RoboDK station: Proyecto 1.rdk

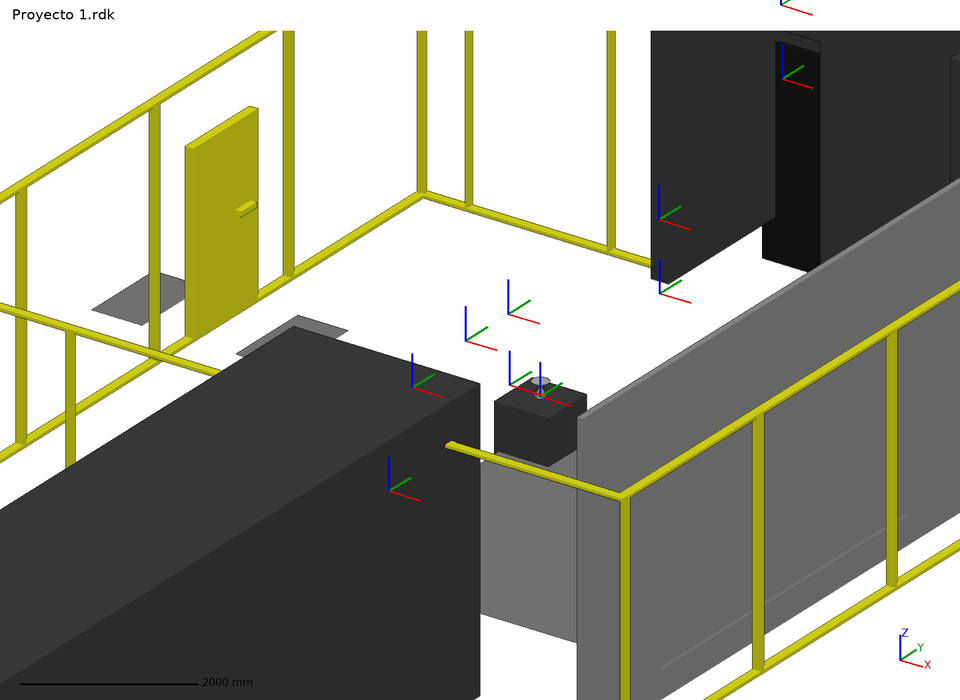
[picture v0: the station drawn from its stored meshes, robots at their saved joint values, targets as dots, program paths as lines]
Station Proyecto (saved by RoboDK 5.8.0). Poses are relative to the parent item; angles as X-Y-Z fixed-axis rotations.
Station parameters (name, value as stored): ColorElegido1, 1, ColorElegido2, 0, Robot1Operando, False, Robot2Operando, False
  - frame ABB IRB 580/12S_2 Base at (840.91, -2530.54, -390.83) mm
    - robot ABB IRB 580/12S 2 (model ABB IRB 580/12S): 6 axes, payload 12 kg, reach 2200 mm, repeatability 0.3 mm, weight 630 kg
        joint limits [-150, -70, -145, -360, -360, -720] to [150, 75, 145, 360, 360, 720]; home [0, 0, 0, 0, 0, 0]; saved at [0, 0, 0, 0, 0, 0]
      - tool TCP2, TCP at (0, -60, 0) mm, geometry from tinker.obj
        - object Herramienta at (0, 0, 0) mm, size 146.3 x 145.2 x 132 mm
        - object Cono at (0, 0, 0) mm, size 720 x 720 x 1182 mm
    - target Pintura21_1 (Cartesian target) at (1116.43, -38.64, 1773.81) mm, rotated rx 90 ry 0 rz 90 deg; joints [-2.419, -0.48, -16.124, 290.45, -28.618, -536.505] of ABB IRB 580/12S 2
    - target Pintura21_2 (Cartesian target) at (1117.91, -195.96, 1412.45) mm, rotated rx 90 ry 89.87 rz 90 deg; joints [-12.073, -6.734, 4.701, 191.643, 22.666, -570.657] of ABB IRB 580/12S 2
    - target Pintura21_3 (Cartesian target) at (1129.28, -196.63, 1042.61) mm, rotated rx 90 ry 89.87 rz 90 deg; joints [-11.969, -2.749, 25.87, 85.216, -50.511, -405.588] of ABB IRB 580/12S 2
    - target Pintura21_4 (Cartesian target) at (1138.7, -115.95, 957.64) mm, rotated rx 176.43 ry 87.92 rz 176.43 deg; joints [-7.055, -0.911, 30.503, 97.258, -52.14, -415.495] of ABB IRB 580/12S 2
    - target Pintura21_5 (Cartesian target) at (1212.31, 299.06, 873.56) mm, rotated rx 176.43 ry 87.92 rz 176.43 deg; joints [16.482, 10.653, 34.896, 146.51, -65.633, -445.211] of ABB IRB 580/12S 2
    - target Pintura21_6 (Cartesian target) at (1200.67, 359.89, 940.4) mm, rotated rx 176.43 ry 87.92 rz 176.43 deg; joints [19.809, 9.031, 31.023, 153.043, -62.201, -454.44] of ABB IRB 580/12S 2
    - target Pintura21_7 (Cartesian target) at (1202.62, 320.47, 971.04) mm, rotated rx 176.43 ry 87.92 rz 176.44 deg; joints [17.751, 7.276, 29.371, 149.237, -57.611, -455.624] of ABB IRB 580/12S 2
    - target Pintura21_8 (Cartesian target) at (1198.4, 183.42, 1272.89) mm, rotated rx 176.44 ry 87.92 rz 176.44 deg; joints [10.425, -0.652, 12.385, 146.399, -25.574, -483.886] of ABB IRB 580/12S 2
    - target Pintura21_9 (Cartesian target) at (1206.42, -176.13, 1230.65) mm, rotated rx 176.44 ry 87.92 rz 176.44 deg; joints [-9.943, 0.129, 14.76, -297.067, -28.151, -41.06] of ABB IRB 580/12S 2
    - target Pintura21_11 (Cartesian target) at (1119.11, -118.32, 1755.25) mm, rotated rx 90 ry 0 rz 90 deg; joints [-7.349, -0.419, -14.975, -51.416, -29.231, -193.501] of ABB IRB 580/12S 2
    - target Pintura21_13 (Cartesian target) at (939.03, -30.25, 1268.55) mm, rotated rx 90 ry 0 rz 90 deg; joints [-2.35, -24.007, 9.647, 83.365, -17.35, -339.315] of ABB IRB 580/12S 2
    - target Pintura21_14 (Cartesian target) at (920.1, -30.25, 1198.47) mm, rotated rx 136.9 ry 0 rz 90 deg; joints [-2.214, -19.899, 6.371, 304.189, -74.383, -511.521] of ABB IRB 580/12S 2
    - target Pintura21_15 (Cartesian target) at (812.29, -30.26, 846.49) mm, rotated rx 90 ry 0 rz 90 deg; joints [-2.837, -28.076, 32.69, 109.612, -58.975, -330.737] of ABB IRB 580/12S 2
    - target Pintura21_16 (Cartesian target) at (926.41, -30.26, 768.39) mm, rotated rx 73.79 ry 0 rz 90 deg; joints [-2.365, -7.019, 46.401, 147.807, -130.027, -297.801] of ABB IRB 580/12S 2
    - target Pintura21_17 (Cartesian target) at (1001.88, -30.25, 1480.86) mm, rotated rx 90 ry 0 rz 90 deg; joints [-2.165, -17.09, -0.641, 345.133, -3.937, -611.896] of ABB IRB 580/12S 2
    - target Pintura21_18 (Cartesian target) at (1001.88, -86.68, 1480.86) mm, rotated rx 90 ry 0 rz 90 deg; joints [-6.183, -16.757, -0.573, 359.165, -10.836, -620.25] of ABB IRB 580/12S 2
    - target Pintura21_19 (Cartesian target) at (1001.88, 52.48, 1480.86) mm, rotated rx 90 ry 0 rz 90 deg; joints [3.753, -16.997, -0.622, 192.113, -6.634, -456.698] of ABB IRB 580/12S 2
    - target Pintura21_20 (Cartesian target) at (1119.11, 44.39, 1755.25) mm, rotated rx 90 ry 0 rz 90 deg; joints [2.77, -0.951, -14.979, 270.402, -26.712, -518.755] of ABB IRB 580/12S 2
    - target Pintura21_21 (Cartesian target) at (1124.85, -28.64, 1773.81) mm, rotated rx 90 ry 0 rz 90 deg; joints [-1.777, 0.178, -16.122, 288.115, -28.472, -534.383] of ABB IRB 580/12S 2
    - target Pintura21_22 (Cartesian target) at (1118.79, 126.71, 1413.18) mm, rotated rx 90 ry 89.87 rz 90 deg; joints [7.867, -7.637, 4.583, 156.485, -15.894, -502.993] of ABB IRB 580/12S 2
    - target Pintura21_23 (Cartesian target) at (1111.66, 131.29, 1043.35) mm, rotated rx 90 ry 89.87 rz 90 deg; joints [8.211, -5.18, 25.707, 128.372, -47.85, -446.42] of ABB IRB 580/12S 2
    - target Pintura21_24 (Cartesian target) at (1116.6, 63.98, 964.01) mm, rotated rx 176.43 ry 87.92 rz 176.43 deg; joints [3.999, -3.356, 30.056, 119.508, -50.327, -436.143] of ABB IRB 580/12S 2
    - target Pintura21_25 (Cartesian target) at (1115.8, -383.46, 874.62) mm, rotated rx 176.43 ry 87.92 rz 176.43 deg; joints [-22.756, 5.765, 35.359, 83.262, -72.027, -389.304] of ABB IRB 580/12S 2
    - target Pintura21_26 (Cartesian target) at (1117.76, -430.8, 936.7) mm, rotated rx 176.43 ry 87.92 rz 176.44 deg; joints [-25.185, 5.256, 31.592, 75.5, -68.929, -384.335] of ABB IRB 580/12S 2
    - target Pintura21_27 (Cartesian target) at (1119.97, -379.27, 974.92) mm, rotated rx 176.43 ry 87.92 rz 176.44 deg; joints [-22.441, 2.586, 29.434, 74.391, -62.633, -387.628] of ABB IRB 580/12S 2
    - target Pintura21_28 (Cartesian target) at (1116.07, -255.92, 1270.03) mm, rotated rx 176.44 ry 87.92 rz 176.44 deg; joints [-15.636, -5.898, 12.34, 45.798, -32.699, -380.627] of ABB IRB 580/12S 2
    - target Pintura21_29 (Cartesian target) at (1113.24, 90.52, 1231.62) mm, rotated rx 176.44 ry 87.92 rz 176.44 deg; joints [5.669, -8.476, 14.275, -235.173, -23.506, -104.543] of ABB IRB 580/12S 2
    - target Pintura21_31 (Cartesian target) at (1117.02, 44.26, 1802.52) mm, rotated rx 90 ry 0 rz 90 deg; joints [2.768, 0.768, -17.925, -85.757, -31.888, -158.337] of ABB IRB 580/12S 2
    - target Pintura21_32 (Cartesian target) at (1119.85, 42.84, 1430.58) mm, rotated rx 90 ry 0 rz 90 deg; joints [2.672, -8.043, 3.565, 130.069, -7.77, -393.618] of ABB IRB 580/12S 2
    - target Pintura21_33 (Cartesian target) at (1113.28, 42.84, 1211.75) mm, rotated rx 90 ry 0 rz 90 deg; joints [2.691, -8.559, 15.797, 111.388, -28.118, -357.829] of ABB IRB 580/12S 2
    - target Pintura21_35 (Cartesian target) at (1350.01, 9.08, 882.74) mm, rotated rx 89.34 ry 0 rz 90 deg; joints [0.453, 17.806, 33.6, 116.92, -61.793, -334.561] of ABB IRB 580/12S 2
    - target Pintura21_34 (Cartesian target) at (1116.39, 45.51, 954.3) mm, rotated rx 78.25 ry 0 rz 90 deg; joints [2.836, -1.144, 33.638, 130.656, -84.724, -326.555] of ABB IRB 580/12S 2
    - target Pintura21_37 (Cartesian target) at (1116.39, -121.21, 954.3) mm, rotated rx 78.25 ry 0 rz 90 deg; joints [-7.514, -0.581, 33.644, 117.012, -85.786, -314.02] of ABB IRB 580/12S 2
    - target Pintura21_36 (Cartesian target) at (1350.01, -80.25, 882.74) mm, rotated rx 89.34 ry 0 rz 90 deg; joints [-3.998, 18.014, 33.552, 109.165, -62.094, -327.854] of ABB IRB 580/12S 2
    - target Pintura21_38 (Cartesian target) at (1113.28, -117.77, 1211.75) mm, rotated rx 90 ry 0 rz 90 deg; joints [-7.362, -8.006, 15.852, 77.337, -30.649, -323.061] of ABB IRB 580/12S 2
    - target Pintura21_39 (Cartesian target) at (1119.85, -118.25, 1430.58) mm, rotated rx 90 ry 0 rz 90 deg; joints [-7.339, -7.506, 3.615, 31.944, -14.28, -290.459] of ABB IRB 580/12S 2
    - target Pintura21_40 (Cartesian target) at (1117.02, -107.51, 1806.84) mm, rotated rx 90 ry 0 rz 90 deg; joints [-6.699, 1.387, -18.207, -55.298, -34.096, -185.427] of ABB IRB 580/12S 2
    - target Pintura22_ 1 (Cartesian target) at (1067.59, 53.4, 1620.15) mm, rotated rx 90 ry 0 rz 90 deg; joints [3.529, -9.086, -7.399, -109.72, -14.309, -148.767] of ABB IRB 580/12S 2
    - target Pintura22_ 2 (Cartesian target) at (1067.59, -94.87, 1462.33) mm, rotated rx 90 ry 0 rz 90 deg; joints [-6.253, -11.629, 1.35, -343.29, -11.164, 82.371] of ABB IRB 580/12S 2
    - target Pintura22_ 3 (Cartesian target) at (1067.59, -259.05, 1472.63) mm, rotated rx 90 ry 0 rz 90 deg; joints [-16.656, -8.853, 1.108, -344.207, -29.317, 98.232] of ABB IRB 580/12S 2
    - target Pintura22_ 4 (Cartesian target) at (1067.59, -164.34, 1317.72) mm, rotated rx 90 ry 0 rz 90 deg; joints [-10.747, -11.653, 9.477, -308.746, -25.051, 58.48] of ABB IRB 580/12S 2
    - target Pintura22_ 5 (Cartesian target) at (1067.59, -224.35, 1182.9) mm, rotated rx 90 ry 0 rz 90 deg; joints [-14.526, -9.793, 17.29, -294.626, -39.656, 55.316] of ABB IRB 580/12S 2
    - target Pintura22_ 6 (Cartesian target) at (1067.59, -116.53, 976.77) mm, rotated rx 90 ry 0 rz 90 deg; joints [-7.665, -7.234, 29.47, -262.498, -54.333, 36.08] of ABB IRB 580/12S 2
    - target Pintura22_ 7 (Cartesian target) at (1067.59, 409.36, 931.57) mm, rotated rx 90 ry 0 rz 90 deg; joints [25.304, 1.291, 32.515, -197.036, -73.881, -2.213] of ABB IRB 580/12S 2
    - target Pintura22_ 8 (Cartesian target) at (1067.59, 392.2, 1026.01) mm, rotated rx 90 ry 0 rz 90 deg; joints [24.369, -2.136, 26.86, -197.594, -64.501, -11.838] of ABB IRB 580/12S 2
    - target Pintura22_ 9 (Cartesian target) at (1067.59, 142.88, 1343.15) mm, rotated rx 90 ry 0 rz 90 deg; joints [9.37, -11.934, 8.012, -211.33, -21.539, -40.301] of ABB IRB 580/12S 2
    - target Pintura22_ 10 (Cartesian target) at (1067.59, -173.83, 1323.16) mm, rotated rx 90 ry 0 rz 90 deg; joints [-11.352, -11.499, 9.193, -310.971, -25.542, 61.091] of ABB IRB 580/12S 2
    - target Pintura22_ 11 (Cartesian target) at (1067.59, 304.45, 953.34) mm, rotated rx 90 ry 0 rz 90 deg; joints [19.372, -2.728, 31.16, -208.004, -65.531, -0.952] of ABB IRB 580/12S 2
    - target Pintura22_ 12 (Cartesian target) at (1137.59, 91.18, 1914.93) mm, rotated rx 110 ry 0 rz 90 deg; joints [5.378, 27.347, -40.85, 26.853, 124.647, -412.723] of ABB IRB 580/12S 2
    - target Pintura22_ 13 (Cartesian target) at (1137.59, 61.18, 1574.93) mm, rotated rx 90 ry 0 rz 90 deg; joints [3.74, -4.471, -4.383, 45.334, 10.05, -323.719] of ABB IRB 580/12S 2
    - target Pintura22_ 14 (Cartesian target) at (1007.59, 0, 1514.93) mm, rotated rx 110 ry 0 rz 90 deg; joints [0, -13.823, -5.955, -70.786, -46.099, -160.785] of ABB IRB 580/12S 2
    - target Pintura22_ 15 (Cartesian target) at (787.59, 0, 1244.93) mm, rotated rx 120 ry 0 rz 90 deg; joints [0, -34.851, 1.653, -68.861, -50.543, -158.857] of ABB IRB 580/12S 2
    - target Pintura22_ 16 (Cartesian target) at (837.59, 0, 784.93) mm, rotated rx 70 ry 0 rz 90 deg; joints [0, -15.633, 44.703, -154.776, 137.797, -244.777] of ABB IRB 580/12S 2
    - target Pintura22_ 17 (Cartesian target) at (1017.59, 50, 784.93) mm, rotated rx 70 ry 0 rz 90 deg; joints [3.455, 0.951, 46.49, -156.092, 146.166, -252.224] of ABB IRB 580/12S 2
    - target Pintura22_ 18 (Cartesian target) at (1017.59, -50, 784.93) mm, rotated rx 70 ry 0 rz 90 deg; joints [-3.456, 0.951, 46.49, -163.171, 146.167, -247.04] of ABB IRB 580/12S 2
    - target Pintura22_ 19 (Cartesian target) at (1057.59, 100, 1214.93) mm, rotated rx 110 ry 0 rz 90 deg; joints [6.572, -12.248, 11.285, -117.423, -18.827, -135.333] of ABB IRB 580/12S 2
    - target Pintura22_ 20 (Cartesian target) at (1057.59, 100, 1304.93) mm, rotated rx 80 ry 0 rz 90 deg; joints [6.641, -12.97, 11.964, -236.168, -40.558, -0.039] of ABB IRB 580/12S 2
    - target Pintura22_ 21 (Cartesian target) at (1137.59, -88.82, 1914.93) mm, rotated rx 110 ry 0 rz 90 deg; joints [-5.239, 27.293, -40.823, 38.325, 124.527, -421.835] of ABB IRB 580/12S 2
    - target Pintura22_ 22 (Cartesian target) at (1137.59, -68.82, 1574.93) mm, rotated rx 90 ry 0 rz 90 deg; joints [-4.206, -4.428, -4.38, 129.57, 10.592, -408.096] of ABB IRB 580/12S 2
    - target Pintura22_ 23 (Cartesian target) at (1057.59, -100, 1214.93) mm, rotated rx 110 ry 0 rz 90 deg; joints [-6.572, -12.248, 11.285, 117.416, 18.825, -404.663] of ABB IRB 580/12S 2
    - target Pintura22_ 24 (Cartesian target) at (1057.59, -100, 1304.93) mm, rotated rx 80 ry 0 rz 90 deg; joints [-6.641, -12.97, 11.964, 236.165, 40.559, -539.963] of ABB IRB 580/12S 2
    - target Pintura22_ 25 (Cartesian target) at (1067.59, -66.6, 1630.15) mm, rotated rx 90 ry 0 rz 90 deg; joints [-4.398, -8.769, -7.95, -54.41, -15.863, -202.263] of ABB IRB 580/12S 2
    - target Pintura22_ 26 (Cartesian target) at (1067.59, 65.12, 1462.33) mm, rotated rx 90 ry 0 rz 90 deg; joints [4.301, -11.851, 1.318, -193.793, -7.847, -69.726] of ABB IRB 580/12S 2
    - target Pintura22_ 27 (Cartesian target) at (1067.59, 230.95, 1472.63) mm, rotated rx 90 ry 0 rz 90 deg; joints [14.935, -9.472, 1.04, -173.077, -26.255, -75.157] of ABB IRB 580/12S 2
    - target Pintura22_ 28 (Cartesian target) at (1067.59, 145.66, 1297.72) mm, rotated rx 90 ry 0 rz 90 deg; joints [9.549, -11.917, 10.56, -217.204, -24.89, -31.418] of ABB IRB 580/12S 2
    - target Pintura22_ 29 (Cartesian target) at (1067.59, 175.65, 1182.9) mm, rotated rx 90 ry 0 rz 90 deg; joints [11.468, -10.727, 17.175, -220.502, -36.246, -17.745] of ABB IRB 580/12S 2
    - target Pintura22_ 30 (Cartesian target) at (1067.59, 73.47, 976.77) mm, rotated rx 90 ry 0 rz 90 deg; joints [4.85, -7.64, 29.432, -237.875, -53.256, 13.804] of ABB IRB 580/12S 2
    - target Pintura22_ 31 (Cartesian target) at (1067.59, -420.64, 931.57) mm, rotated rx 90 ry 0 rz 90 deg; joints [-25.911, 1.686, 32.507, -280.163, -74.568, 66.389] of ABB IRB 580/12S 2
    - target Pintura22_ 32 (Cartesian target) at (1067.59, -477.8, 1006.02) mm, rotated rx 90 ry 0 rz 90 deg; joints [-28.891, 1.54, 28.051, -288.806, -71.996, 72.955] of ABB IRB 580/12S 2
    - target Pintura22_ 33 (Cartesian target) at (1067.59, -187.12, 1323.15) mm, rotated rx 90 ry 0 rz 90 deg; joints [-12.194, -11.273, 9.224, -312.414, -26.747, 63.467] of ABB IRB 580/12S 2
    - target Pintura22_ 34 (Cartesian target) at (1067.59, 96.17, 1323.16) mm, rotated rx 90 ry 0 rz 90 deg; joints [6.338, -12.498, 9.051, -226.848, -19.298, -26.794] of ABB IRB 580/12S 2
    - target Pintura22_ 35 (Cartesian target) at (1067.59, -325.55, 953.34) mm, rotated rx 90 ry 0 rz 90 deg; joints [-20.605, -2.127, 31.178, -277.633, -66.76, 58.537] of ABB IRB 580/12S 2
    - target Pintura22_ 36 (Cartesian target) at (1236.43, -90.2, 1853.81) mm, rotated rx 109.13 ry 0 rz 90 deg; joints [-4.929, 20.785, -28.819, 315.941, -90.742, -506.111] of ABB IRB 580/12S 2
    - target Pintura22_ 37 (Cartesian target) at (1012.5, -90.2, 1474.16) mm, rotated rx 90.64 ry 0 rz 90 deg; joints [-6.348, -15.932, -0.16, 357.376, -11.167, -618.246] of ABB IRB 580/12S 2
    - target Pintura22_ 38 (Cartesian target) at (1094.1, -119.86, 1001.32) mm, rotated rx 90.64 ry 0 rz 90 deg; joints [-7.65, -5.739, 28.002, 232.585, 50.499, -546.78] of ABB IRB 580/12S 2
    - target Pintura22_ 39 (Cartesian target) at (1389.03, -96.9, 885.54) mm, rotated rx 83 ry 0 rz 90 deg; joints [-4.66, 21.788, 33.785, 230.644, 75.314, -566.392] of ABB IRB 580/12S 2
    - target Pintura22_ 40 (Cartesian target) at (1389.03, 71.9, 885.55) mm, rotated rx 83 ry 0 rz 90 deg; joints [3.461, 21.655, 33.821, 243.013, 75.168, -576.616] of ABB IRB 580/12S 2
    - target Pintura22_ 41 (Cartesian target) at (1094.1, 98.81, 1001.32) mm, rotated rx 90.64 ry 0 rz 90 deg; joints [6.318, -5.957, 27.986, 262.69, 49.904, -572.808] of ABB IRB 580/12S 2
    - target Pintura22_ 42 (Cartesian target) at (1012.5, 114.28, 1474.16) mm, rotated rx 90.64 ry 0 rz 90 deg; joints [8.023, -15.687, -0.113, 191.161, -14.073, -449.577] of ABB IRB 580/12S 2
    - target Pintura22_ 43 (Cartesian target) at (1236.43, 75.05, 1853.81) mm, rotated rx 109.13 ry 0 rz 90 deg; joints [4.104, 20.635, -28.772, 304.34, -90.475, -495.607] of ABB IRB 580/12S 2
    - target Pintura22_ 44 (Cartesian target) at (1208.68, -23.31, 1762.17) mm, rotated rx 90.64 ry 0 rz 90 deg; joints [-1.326, 6.871, -15.851, 286.646, -29.056, -532.5] of ABB IRB 580/12S 2
    - target Pintura22_ 45 (Cartesian target) at (1286.9, -13.32, 1041.23) mm, rotated rx 90.64 ry 0 rz 90 deg; joints [-0.703, 8.327, 25.435, 106.626, -43.976, -340.184] of ABB IRB 580/12S 2
    - target Pintura22_ 46 (Cartesian target) at (1224.34, -13.32, 1041.93) mm, rotated rx 90.64 ry 0.07 rz 83.59 deg; joints [0.515, 3.407, 25.753, 125.206, -46.158, -355.175] of ABB IRB 580/12S 2
    - target Pintura22_ 47 (Cartesian target) at (1230.82, -13.31, 1620.47) mm, rotated rx 90.64 ry 0.07 rz 83.59 deg; joints [0.511, 4.181, -7.144, 235.62, -18.187, -491.147] of ABB IRB 580/12S 2
    - target Pintura22_ 48 (Cartesian target) at (1230.82, -13.31, 1620.47) mm, rotated rx 90.63 ry -0.13 rz 101.88 deg; joints [-3.038, 4.556, -7.162, 345.144, -29.508, -589.807] of ABB IRB 580/12S 2
    - target Pintura22_ 49 (Cartesian target) at (1224, -13.32, 1012.28) mm, rotated rx 90.63 ry -0.13 rz 101.88 deg; joints [-3.058, 4.47, 27.441, 216.544, 54.407, -535.823] of ABB IRB 580/12S 2
    - object peana at (0, 0, -390) mm, rotated rx 90 ry 0 rz 0 deg, size 750 x 750 x 750 mm, 998277249 curves, geometry from peana.obj
  - frame ABB IRB 580/12S_1 Base at (840.91, 429.46, -390.83) mm
    - robot ABB IRB 580/12S 1 (model ABB IRB 580/12S): 6 axes, payload 12 kg, reach 2200 mm, repeatability 0.3 mm, weight 630 kg
        joint limits [-150, -70, -145, -360, -360, -720] to [150, 75, 145, 360, 360, 720]; home [0, 0, 0, 0, 0, 0]; saved at [-2.419, -0.48, -16.124, 290.45, -28.618, -176.505]
      - tool TCP1, TCP at (0, 0, 0) mm, geometry from tinker.obj
        - object Herramienta at (0, 0, 0) mm, size 146.3 x 145.2 x 132 mm
    - target Pintura11_1 (Cartesian target) at (1116.43, -38.64, 1773.81) mm, rotated rx 90 ry 0 rz 90 deg; joints [-2.419, -0.48, -16.124, 290.45, -28.618, -536.505] of ABB IRB 580/12S 1
    - target Pintura11_2 (Cartesian target) at (1117.91, -195.96, 1412.45) mm, rotated rx 90 ry 89.87 rz 90 deg; joints [-12.073, -6.734, 4.701, 191.643, 22.666, -570.657] of ABB IRB 580/12S 1
    - target Pintura11_3 (Cartesian target) at (1129.28, -196.63, 1042.61) mm, rotated rx 90 ry 89.87 rz 90 deg; joints [-11.969, -2.749, 25.87, 85.216, -50.511, -405.588] of ABB IRB 580/12S 1
    - target Pintura11_4 (Cartesian target) at (1138.7, -115.95, 957.64) mm, rotated rx 176.43 ry 87.92 rz 176.43 deg; joints [-7.055, -0.911, 30.503, 97.258, -52.14, -415.495] of ABB IRB 580/12S 1
    - target Pintura11_5 (Cartesian target) at (1212.31, 299.06, 873.56) mm, rotated rx 176.43 ry 87.92 rz 176.43 deg; joints [16.482, 10.653, 34.896, 146.51, -65.633, -445.211] of ABB IRB 580/12S 1
    - target Pintura11_6 (Cartesian target) at (1200.67, 359.89, 940.4) mm, rotated rx 176.43 ry 87.92 rz 176.43 deg; joints [19.809, 9.031, 31.023, 153.043, -62.201, -454.44] of ABB IRB 580/12S 1
    - target Pintura11_7 (Cartesian target) at (1202.62, 320.47, 971.04) mm, rotated rx 176.43 ry 87.92 rz 176.44 deg; joints [17.751, 7.276, 29.371, 149.237, -57.611, -455.624] of ABB IRB 580/12S 1
    - target Pintura11_8 (Cartesian target) at (1198.4, 183.42, 1272.89) mm, rotated rx 176.44 ry 87.92 rz 176.44 deg; joints [10.425, -0.652, 12.385, 146.399, -25.574, -483.886] of ABB IRB 580/12S 1
    - target Pintura11_9 (Cartesian target) at (1206.42, -176.13, 1230.65) mm, rotated rx 176.44 ry 87.92 rz 176.44 deg; joints [-9.943, 0.129, 14.76, -297.067, -28.151, -41.06] of ABB IRB 580/12S 1
    - target Pintura11_11 (Cartesian target) at (1119.11, -118.32, 1755.25) mm, rotated rx 90 ry 0 rz 90 deg; joints [-7.349, -0.419, -14.975, -51.416, -29.231, -193.501] of ABB IRB 580/12S 1
    - target Pintura11_13 (Cartesian target) at (939.03, -30.25, 1268.55) mm, rotated rx 90 ry 0 rz 90 deg; joints [-2.35, -24.007, 9.647, 83.365, -17.35, -339.315] of ABB IRB 580/12S 1
    - target Pintura11_14 (Cartesian target) at (920.1, -30.25, 1198.47) mm, rotated rx 136.9 ry 0 rz 90 deg; joints [-2.214, -19.899, 6.371, 304.189, -74.383, -511.521] of ABB IRB 580/12S 1
    - target Pintura11_15 (Cartesian target) at (812.29, -30.26, 846.49) mm, rotated rx 90 ry 0 rz 90 deg; joints [-2.837, -28.076, 32.69, 109.612, -58.975, -330.737] of ABB IRB 580/12S 1
    - target Pintura11_16 (Cartesian target) at (926.41, -30.26, 768.39) mm, rotated rx 73.79 ry 0 rz 90 deg; joints [-2.365, -7.019, 46.401, 147.807, -130.027, -297.801] of ABB IRB 580/12S 1
    - target Pintura11_17 (Cartesian target) at (1001.88, -30.25, 1480.86) mm, rotated rx 90 ry 0 rz 90 deg; joints [-2.165, -17.09, -0.641, 345.133, -3.937, -611.896] of ABB IRB 580/12S 1
    - target Pintura11_18 (Cartesian target) at (1001.88, -86.68, 1480.86) mm, rotated rx 90 ry 0 rz 90 deg; joints [-6.183, -16.757, -0.573, 359.165, -10.836, -620.25] of ABB IRB 580/12S 1
    - target Pintura11_19 (Cartesian target) at (1001.88, 52.48, 1480.86) mm, rotated rx 90 ry 0 rz 90 deg; joints [3.753, -16.997, -0.622, 192.113, -6.634, -456.698] of ABB IRB 580/12S 1
    - target Pintura11_20 (Cartesian target) at (1119.11, 44.39, 1755.25) mm, rotated rx 90 ry 0 rz 90 deg; joints [2.77, -0.951, -14.979, 270.402, -26.712, -518.755] of ABB IRB 580/12S 1
    - target Pintura12_1 (Cartesian target) at (1067.59, 13.4, 1620.15) mm, rotated rx 90 ry 0 rz 90 deg; joints [0.887, -9.208, -7.413, -91.494, -13.034, -167.871] of ABB IRB 580/12S 1
    - target Pintura12_2 (Cartesian target) at (1067.59, -94.87, 1462.33) mm, rotated rx 90 ry 0 rz 90 deg; joints [-6.253, -11.629, 1.35, -343.29, -11.164, 82.371] of ABB IRB 580/12S 1
    - target Pintura12_3 (Cartesian target) at (1067.59, -259.05, 1472.63) mm, rotated rx 90 ry 0 rz 90 deg; joints [-16.656, -8.853, 1.108, -344.207, -29.317, 98.232] of ABB IRB 580/12S 1
    - target Pintura12_4 (Cartesian target) at (1067.59, -224.34, 1297.72) mm, rotated rx 90 ry 0 rz 90 deg; joints [-14.526, -10.541, 10.744, -311.194, -31.651, 65.963] of ABB IRB 580/12S 1
    - target Pintura12_5 (Cartesian target) at (1067.59, -224.35, 1182.9) mm, rotated rx 90 ry 0 rz 90 deg; joints [-14.526, -9.793, 17.29, -294.626, -39.656, 55.316] of ABB IRB 580/12S 1
    - target Pintura12_6 (Cartesian target) at (1067.59, -116.53, 976.77) mm, rotated rx 90 ry 0 rz 90 deg; joints [-7.665, -7.234, 29.47, -262.498, -54.333, 36.08] of ABB IRB 580/12S 1
    - target Pintura12_7 (Cartesian target) at (1067.59, 389.36, 931.57) mm, rotated rx 90 ry 0 rz 90 deg; joints [24.212, 0.61, 32.523, -199.021, -72.671, -1.681] of ABB IRB 580/12S 1
    - target Pintura12_8 (Cartesian target) at (1067.59, 382.2, 1006.01) mm, rotated rx 90 ry 0 rz 90 deg; joints [23.817, -1.941, 28.042, -199.018, -65.5, -9.384] of ABB IRB 580/12S 1
    - target Pintura12_9 (Cartesian target) at (1067.59, 122.88, 1323.15) mm, rotated rx 90 ry 0 rz 90 deg; joints [8.078, -12.217, 9.092, -219.336, -21.246, -32.553] of ABB IRB 580/12S 1
    - target Pintura12_10 (Cartesian target) at (1067.59, -173.83, 1323.16) mm, rotated rx 90 ry 0 rz 90 deg; joints [-11.352, -11.499, 9.193, -310.971, -25.542, 61.091] of ABB IRB 580/12S 1
    - target Pintura12_11 (Cartesian target) at (1067.59, 274.45, 953.34) mm, rotated rx 90 ry 0 rz 90 deg; joints [17.587, -3.524, 31.128, -211.447, -63.849, 0.455] of ABB IRB 580/12S 1
    - target Pintura12_37 (Cartesian target) at (1236.43, -90.2, 1853.81) mm, rotated rx 109.13 ry 0 rz 90 deg; joints [-4.929, 20.785, -28.819, 315.941, -90.742, -506.111] of ABB IRB 580/12S 1
    - target Pintura12_38 (Cartesian target) at (1012.5, -90.2, 1474.16) mm, rotated rx 90.64 ry 0 rz 90 deg; joints [-6.348, -15.932, -0.16, 357.376, -11.167, -618.246] of ABB IRB 580/12S 1
    - target Pintura12_39 (Cartesian target) at (1094.1, -119.86, 1001.32) mm, rotated rx 90.64 ry 0 rz 90 deg; joints [-7.65, -5.739, 28.002, 232.585, 50.499, -546.78] of ABB IRB 580/12S 1
    - target Pintura12_40 (Cartesian target) at (1389.03, -96.9, 885.54) mm, rotated rx 83 ry 0 rz 90 deg; joints [-4.66, 21.788, 33.785, 230.644, 75.314, -566.392] of ABB IRB 580/12S 1
    - target Pintura12_41 (Cartesian target) at (1389.03, 71.9, 885.55) mm, rotated rx 83 ry 0 rz 90 deg; joints [3.461, 21.655, 33.821, 243.013, 75.168, -576.616] of ABB IRB 580/12S 1
    - target Pintura12_42 (Cartesian target) at (1094.1, 98.81, 1001.32) mm, rotated rx 90.64 ry 0 rz 90 deg; joints [6.318, -5.957, 27.986, 262.69, 49.904, -572.808] of ABB IRB 580/12S 1
    - target Pintura12_43 (Cartesian target) at (1012.5, 114.28, 1474.16) mm, rotated rx 90.64 ry 0 rz 90 deg; joints [8.023, -15.687, -0.113, 191.161, -14.073, -449.577] of ABB IRB 580/12S 1
    - target Pintura12_44 (Cartesian target) at (1236.43, 75.05, 1853.81) mm, rotated rx 109.13 ry 0 rz 90 deg; joints [4.104, 20.635, -28.772, 304.34, -90.475, -495.607] of ABB IRB 580/12S 1
    - target Pintura12_45 (Cartesian target) at (1208.68, -23.31, 1762.17) mm, rotated rx 90.64 ry 0 rz 90 deg; joints [-1.326, 6.871, -15.851, 286.646, -29.056, -532.5] of ABB IRB 580/12S 1
    - target Pintura12_46 (Cartesian target) at (1286.9, -13.32, 1041.23) mm, rotated rx 90.64 ry 0 rz 90 deg; joints [-0.703, 8.327, 25.435, 106.626, -43.976, -340.184] of ABB IRB 580/12S 1
    - target Pintura12_47 (Cartesian target) at (1224.34, -13.32, 1041.93) mm, rotated rx 90.64 ry 0.07 rz 83.59 deg; joints [0.515, 3.407, 25.753, 125.206, -46.158, -355.175] of ABB IRB 580/12S 1
    - target Pintura12_48 (Cartesian target) at (1230.82, -13.31, 1620.47) mm, rotated rx 90.64 ry 0.07 rz 83.59 deg; joints [0.511, 4.181, -7.144, 235.62, -18.187, -491.147] of ABB IRB 580/12S 1
    - target Pintura12_49 (Cartesian target) at (1230.82, -13.31, 1620.47) mm, rotated rx 90.63 ry -0.13 rz 101.88 deg; joints [-3.038, 4.556, -7.162, 345.144, -29.508, -589.807] of ABB IRB 580/12S 1
    - target Pintura12_50 (Cartesian target) at (1224, -13.32, 1012.28) mm, rotated rx 90.63 ry -0.13 rz 101.88 deg; joints [-3.058, 4.47, 27.441, 216.544, 54.407, -535.823] of ABB IRB 580/12S 1
    - target Pintura11_21 (Cartesian target) at (1124.85, -18.64, 1773.81) mm, rotated rx 90 ry 0 rz 90 deg; joints [-1.157, 0.157, -16.122, 285.858, -28.374, -532.295] of ABB IRB 580/12S 1
    - target Pintura11_22 (Cartesian target) at (1118.79, 126.71, 1413.18) mm, rotated rx 90 ry 89.87 rz 90 deg; joints [7.867, -7.637, 4.583, 156.485, -15.894, -502.993] of ABB IRB 580/12S 1
    - target Pintura11_23 (Cartesian target) at (1111.66, 131.29, 1043.35) mm, rotated rx 90 ry 89.87 rz 90 deg; joints [8.211, -5.18, 25.707, 128.372, -47.85, -446.42] of ABB IRB 580/12S 1
    - target Pintura11_24 (Cartesian target) at (1116.6, 63.98, 964.01) mm, rotated rx 176.43 ry 87.92 rz 176.43 deg; joints [3.999, -3.356, 30.056, 119.508, -50.327, -436.143] of ABB IRB 580/12S 1
    - target Pintura11_25 (Cartesian target) at (1115.8, -383.46, 874.62) mm, rotated rx 176.43 ry 87.92 rz 176.43 deg; joints [-22.756, 5.765, 35.359, 83.262, -72.027, -389.304] of ABB IRB 580/12S 1
    - target Pintura11_26 (Cartesian target) at (1117.76, -430.8, 936.7) mm, rotated rx 176.43 ry 87.92 rz 176.44 deg; joints [-25.185, 5.256, 31.592, 75.5, -68.929, -384.335] of ABB IRB 580/12S 1
    - target Pintura11_27 (Cartesian target) at (1119.97, -379.27, 974.92) mm, rotated rx 176.43 ry 87.92 rz 176.44 deg; joints [-22.441, 2.586, 29.434, 74.391, -62.633, -387.628] of ABB IRB 580/12S 1
    - target Pintura11_28 (Cartesian target) at (1116.07, -255.92, 1270.03) mm, rotated rx 176.44 ry 87.92 rz 176.44 deg; joints [-15.636, -5.898, 12.34, 45.798, -32.699, -380.627] of ABB IRB 580/12S 1
    - target Pintura11_29 (Cartesian target) at (1113.24, 90.52, 1231.62) mm, rotated rx 176.44 ry 87.92 rz 176.44 deg; joints [5.669, -8.476, 14.275, -235.173, -23.506, -104.543] of ABB IRB 580/12S 1
    - target Pintura11_31 (Cartesian target) at (1117.02, 44.26, 1802.52) mm, rotated rx 90 ry 0 rz 90 deg; joints [2.768, 0.768, -17.925, -85.757, -31.888, -158.337] of ABB IRB 580/12S 1
    - target Pintura11_32 (Cartesian target) at (1119.85, 42.84, 1430.58) mm, rotated rx 90 ry 0 rz 90 deg; joints [2.672, -8.043, 3.565, 130.069, -7.77, -393.618] of ABB IRB 580/12S 1
    - target Pintura11_33 (Cartesian target) at (1113.28, 42.84, 1211.75) mm, rotated rx 90 ry 0 rz 90 deg; joints [2.691, -8.559, 15.797, 111.388, -28.118, -357.829] of ABB IRB 580/12S 1
    - target Pintura11_35 (Cartesian target) at (1350.01, 9.08, 882.74) mm, rotated rx 89.34 ry 0 rz 90 deg; joints [0.453, 17.806, 33.6, 116.92, -61.793, -334.561] of ABB IRB 580/12S 1
    - target Pintura11_34 (Cartesian target) at (1116.39, 45.51, 954.3) mm, rotated rx 78.25 ry 0 rz 90 deg; joints [2.836, -1.144, 33.638, 130.656, -84.724, -326.555] of ABB IRB 580/12S 1
    - target Pintura11_37 (Cartesian target) at (1116.39, -121.21, 954.3) mm, rotated rx 78.25 ry 0 rz 90 deg; joints [-7.514, -0.581, 33.644, 117.012, -85.786, -314.02] of ABB IRB 580/12S 1
    - target Pintura11_36 (Cartesian target) at (1350.01, -80.25, 882.74) mm, rotated rx 89.34 ry 0 rz 90 deg; joints [-3.998, 18.014, 33.552, 109.165, -62.094, -327.854] of ABB IRB 580/12S 1
    - target Pintura11_38 (Cartesian target) at (1113.28, -117.77, 1211.75) mm, rotated rx 90 ry 0 rz 90 deg; joints [-7.362, -8.006, 15.852, 77.337, -30.649, -323.061] of ABB IRB 580/12S 1
    - target Pintura11_39 (Cartesian target) at (1119.85, -118.25, 1430.58) mm, rotated rx 90 ry 0 rz 90 deg; joints [-7.339, -7.506, 3.615, 31.944, -14.28, -290.459] of ABB IRB 580/12S 1
    - target Pintura11_40 (Cartesian target) at (1117.02, -107.51, 1806.84) mm, rotated rx 90 ry 0 rz 90 deg; joints [-6.699, 1.387, -18.207, -55.298, -34.096, -185.427] of ABB IRB 580/12S 1
    - target Pintura12_13 (Cartesian target) at (1137.59, 91.18, 1934.93) mm, rotated rx 110 ry 0 rz 90 deg; joints [5.494, 17.782, -34.165, 36.405, 105.718, -401.654] of ABB IRB 580/12S 1
    - target Pintura12_14 (Cartesian target) at (1137.59, 61.18, 1574.93) mm, rotated rx 90 ry 0 rz 90 deg; joints [3.74, -4.471, -4.383, 45.334, 10.05, -323.719] of ABB IRB 580/12S 1
    - target Pintura12_15 (Cartesian target) at (1007.59, 0, 1514.93) mm, rotated rx 110 ry 0 rz 90 deg; joints [0, -13.823, -5.955, -70.786, -46.099, -160.785] of ABB IRB 580/12S 1
    - target Pintura12_16 (Cartesian target) at (787.59, 0, 1244.93) mm, rotated rx 120 ry 0 rz 90 deg; joints [0, -34.851, 1.653, -68.861, -50.543, -158.857] of ABB IRB 580/12S 1
    - target Pintura12_17 (Cartesian target) at (837.59, 0, 784.93) mm, rotated rx 70 ry 0 rz 90 deg; joints [0, -15.633, 44.703, -154.776, 137.797, -244.777] of ABB IRB 580/12S 1
    - target Pintura12_18 (Cartesian target) at (1017.59, 50, 784.93) mm, rotated rx 70 ry 0 rz 90 deg; joints [3.455, 0.951, 46.49, -156.092, 146.166, -252.224] of ABB IRB 580/12S 1
    - target Pintura12_19 (Cartesian target) at (1017.59, -50, 784.93) mm, rotated rx 70 ry 0 rz 90 deg; joints [-3.456, 0.951, 46.49, -163.171, 146.167, -247.04] of ABB IRB 580/12S 1
    - target Pintura12_20 (Cartesian target) at (1057.59, 100, 1214.93) mm, rotated rx 110 ry 0 rz 90 deg; joints [6.572, -12.248, 11.285, -117.423, -18.827, -135.333] of ABB IRB 580/12S 1
    - target Pintura12_21 (Cartesian target) at (1057.59, 100, 1304.93) mm, rotated rx 80 ry 0 rz 90 deg; joints [6.641, -12.97, 11.964, -236.168, -40.558, -0.039] of ABB IRB 580/12S 1
    - target Pintura12_22 (Cartesian target) at (1137.59, -88.82, 1934.93) mm, rotated rx 110 ry 0 rz 90 deg; joints [-5.352, 17.754, -34.157, 48.973, 105.665, -412.663] of ABB IRB 580/12S 1
    - target Pintura12_23 (Cartesian target) at (1137.59, -68.82, 1574.93) mm, rotated rx 90 ry 0 rz 90 deg; joints [-4.206, -4.428, -4.38, 129.57, 10.592, -408.096] of ABB IRB 580/12S 1
    - target Pintura12_24 (Cartesian target) at (1057.59, -100, 1214.93) mm, rotated rx 110 ry 0 rz 90 deg; joints [-6.572, -12.248, 11.285, 117.416, 18.825, -404.663] of ABB IRB 580/12S 1
    - target Pintura12_25 (Cartesian target) at (1057.59, -100, 1304.93) mm, rotated rx 80 ry 0 rz 90 deg; joints [-6.641, -12.97, 11.964, 236.165, 40.559, -539.963] of ABB IRB 580/12S 1
    - target Pintura12_26 (Cartesian target) at (1067.59, -26.6, 1760.15) mm, rotated rx 90 ry 0 rz 90 deg; joints [-1.76, -4.948, -15.437, -72.183, -27.257, -175.112] of ABB IRB 580/12S 1
    - target Pintura12_27 (Cartesian target) at (1067.59, 65.12, 1462.33) mm, rotated rx 90 ry 0 rz 90 deg; joints [4.301, -11.851, 1.318, -193.793, -7.847, -69.726] of ABB IRB 580/12S 1
    - target Pintura12_28 (Cartesian target) at (1067.59, 230.95, 1472.63) mm, rotated rx 90 ry 0 rz 90 deg; joints [14.935, -9.472, 1.04, -173.077, -26.255, -75.157] of ABB IRB 580/12S 1
    - target Pintura12_29 (Cartesian target) at (1067.59, 145.66, 1297.72) mm, rotated rx 90 ry 0 rz 90 deg; joints [9.549, -11.917, 10.56, -217.204, -24.89, -31.418] of ABB IRB 580/12S 1
    - target Pintura12_30 (Cartesian target) at (1067.59, 175.65, 1182.9) mm, rotated rx 90 ry 0 rz 90 deg; joints [11.468, -10.727, 17.175, -220.502, -36.246, -17.745] of ABB IRB 580/12S 1
    - target Pintura12_31 (Cartesian target) at (1067.59, 73.47, 976.77) mm, rotated rx 90 ry 0 rz 90 deg; joints [4.85, -7.64, 29.432, -237.875, -53.256, 13.804] of ABB IRB 580/12S 1
    - target Pintura12_32 (Cartesian target) at (1067.59, -420.64, 931.57) mm, rotated rx 90 ry 0 rz 90 deg; joints [-25.911, 1.686, 32.507, -280.163, -74.568, 66.389] of ABB IRB 580/12S 1
    - target Pintura12_33 (Cartesian target) at (1067.59, -477.8, 1006.02) mm, rotated rx 90 ry 0 rz 90 deg; joints [-28.891, 1.54, 28.051, -288.806, -71.996, 72.955] of ABB IRB 580/12S 1
    - target Pintura12_34 (Cartesian target) at (1067.59, -187.12, 1323.15) mm, rotated rx 90 ry 0 rz 90 deg; joints [-12.194, -11.273, 9.224, -312.414, -26.747, 63.467] of ABB IRB 580/12S 1
    - target Pintura12_35 (Cartesian target) at (1067.59, 96.17, 1323.16) mm, rotated rx 90 ry 0 rz 90 deg; joints [6.338, -12.498, 9.051, -226.848, -19.298, -26.794] of ABB IRB 580/12S 1
    - target Pintura12_36 (Cartesian target) at (1067.59, -325.55, 953.34) mm, rotated rx 90 ry 0 rz 90 deg; joints [-20.605, -2.127, 31.178, -277.633, -66.76, 58.537] of ABB IRB 580/12S 1
    - object peana at (0, 0, -390) mm, rotated rx 90 ry 0 rz 0 deg, size 750 x 750 x 750 mm, 998277249 curves, geometry from peana.obj
  - frame Frame Grua at (2500, -3400.54, 2300) mm
    - object grua at (0, 0, 0) mm, rotated rx 90 ry 0 rz 0 deg, size 0 x 0 x 0 mm, 1044167869 curves, geometry from grua.obj
  - frame Frame 8 at (0, -870.54, 0) mm
    - object Fabrica 1 at (0, 0, -1030) mm, rotated rx 90 ry 0 rz 0 deg
    - object Pasillo 2 at (4600, 16100, -1460) mm, rotated rx 90 ry 0 rz 90 deg, size 20643.2 x 3904.4 x 2560.3 mm, geometry from Pasillo 2.obj
    - object Pasillo 2 at (500, 16100, -1460) mm, rotated rx 90 ry 0 rz 90 deg, size 20643.2 x 3904.4 x 2560.3 mm, geometry from Pasillo 2.obj
    - object Pasillo 2 at (2500, -14400, -1460) mm, rotated rx 90 ry 0 rz 90 deg, size 20643.2 x 3904.4 x 2560.3 mm, geometry from Pasillo 2.obj
    - object Valla 2 at (-200, 0, 0) mm, rotated rx 0 ry 0 rz -90 deg, size 120 x 3276.4 x 2628 mm, geometry from Valla 2.obj
    - object Valla 2 at (1450, -8420, 0) mm, size 120 x 3276.4 x 2628 mm, geometry from Valla 2.obj
    - object Valla 2 at (1450, -5800, 0) mm, size 120 x 3276.4 x 2628 mm, geometry from Valla 2.obj
    - object Valla 2 at (2180, -1330, 0) mm, rotated rx 0 ry 0 rz 10 deg, size 120 x 3276.4 x 2628 mm, geometry from Valla 2.obj
    - object Valla 2 at (1450, -3180, 0) mm, size 120 x 3276.4 x 2628 mm, geometry from Valla 2.obj
    - object Valla 2 at (-5180, 0, 0) mm, rotated rx 0 ry 0 rz -90 deg, size 120 x 3276.4 x 2628 mm, geometry from Valla 2.obj
    - object Valla 2 at (-8660, -8420, 0) mm, size 120 x 3276.4 x 2628 mm, geometry from Valla 2.obj
    - object Valla 2 at (-7800, 0, 0) mm, rotated rx 0 ry 0 rz -90 deg, size 120 x 3276.4 x 2628 mm, geometry from Valla 2.obj
    - object Valla 2 at (-8660, -5800, 0) mm, size 120 x 3276.4 x 2628 mm, geometry from Valla 2.obj
    - object Valla 3 at (-3960, 1910, -1030) mm, rotated rx 90 ry 0 rz 0 deg, size 284.8 x 3276.4 x 2628 mm, geometry from Valla 3.obj
    - object Valla 2 at (-7760, 10540, 0) mm, rotated rx 0 ry 0 rz -90 deg, size 120 x 3276.4 x 2628 mm, geometry from Valla 2.obj
    - object Valla 2 at (-8660, -560, 0) mm, size 120 x 3276.4 x 2628 mm, geometry from Valla 2.obj
    - object Valla 2 at (-7110, 10540, 0) mm, rotated rx 0 ry 0 rz -90 deg, size 120 x 3276.4 x 2628 mm, geometry from Valla 2.obj
    - object IRONLINELOGOChasis at (-460, 0, 0) mm, size 4826 x 4699 x 0 mm, 1046087008 curves, geometry from IRONLINELOGOChasis.png
    - object pared at (-500, 0, 0) mm, size 83.4 x 3742.7 x 4117 mm, geometry from pared.obj
    - object pared at (-500, 0, 0) mm, size 83.4 x 3742.7 x 4117 mm, geometry from pared.obj
    - object IronLineFUll text at (0, 0, 0) mm, size 5022.9 x 2070.1 x 0 mm, 1046086528 curves, geometry from IronLineFUll text.png
    - object pared at (0, 0, 0) mm, size 2495.2 x 55.6 x 2744.6 mm
    - object pared at (1960, -13550, 0) mm, size 2495.2 x 55.6 x 2744.6 mm
    - object pared at (4100, 0, 0) mm, size 2495.2 x 55.6 x 2744.6 mm
    - object Flecha at (-330, 0, 0) mm, size 1219.2 x 693.6 x 0 mm, 1046083728 curves, geometry from Flecha.png
    - object Flecha at (-7590, 3760, 0) mm, rotated rx 0 ry 0 rz -180 deg, size 1219.2 x 693.6 x 0 mm, 1046083728 curves, geometry from Flecha.png
    - object Ralla at (-1300, -160, -1020) mm
    - object pared at (13600, 0, 0) mm, size 83.4 x 3742.7 x 4117 mm, geometry from pared.obj
  - frame Frame 6 at (2490.38, -2530.4, 1393.84) mm
    - object Chopper Frame AP203 2 at (-5, -165, -630) mm, rotated rx 0 ry -90 rz 0 deg
  - frame Frame C1 at (4518.72, 5642.83, 2280.87) mm
    - object Cilindro2 at (-60, 0, -830) mm, rotated rx 0 ry 4.5 rz 0 deg
  - frame Frame H1 at (2478.72, 415.5, 2280.87) mm
    - object Cilindro2 at (-60, 0, -830) mm, rotated rx 0 ry 4.5 rz 0 deg
  - frame Frame 4 at (4530.38, 5646.93, 1393.84) mm
    - object Chopper Frame AP203 1 at (-5, -165, -630) mm, rotated rx 0 ry -90 rz 0 deg
  - frame Frame 5 at (2485.91, 420, 1357.58) mm
    - object Frame cb 750 1 at (0, -127.82, -424.28) mm, rotated rx 90 ry -70 rz -90 deg
  - frame Frame C2 at (2478.72, -2534.5, 2280.87) mm
    - object Cilindro3 at (-60, 0, -830) mm, rotated rx 0 ry 4.5 rz 0 deg
  - frame Frame H2 at (448.72, 5708.5, 2280.87) mm
    - object Cilindro2 at (-60, 0, -830) mm, rotated rx 0 ry 4.5 rz 0 deg
  - frame Frame 7 at (455.92, 5713, 1357.58) mm
    - object Frame cb 750 2 at (0, -127.82, -424.28) mm, rotated rx 90 ry -70 rz -90 deg
  - folder Programas
    - Python program Honda11 (listed below)
    - Python program Honda12 (listed below)
    - Python program Chopper11 (listed below)
    - Python program Chopper12 (listed below)
    - Python program Honda21 (listed below)
    - Python program Honda22 (listed below)
    - Python program Chopper21 (listed below)
    - Python program Chopper22 (listed below)
    - Python program SprayOn (listed below)
    - Python program MoverHonda11 (listed below)
    - Python program MoverHonda12 (listed below)
    - Python program MoverChopper11 (listed below)
    - Python program MoverChopper12 (listed below)
    - Python program MoverHonda21 (listed below)
    - Python program MoverHonda22 (listed below)
    - Python program MoverChopper21 (listed below)
    - Python program MoverChopper22 (listed below)
    - Python program MoverChopper11Final (listed below)
    - Python program MoverChopper12Final (listed below)
    - Python program MoverHonda11Final (listed below)
    - Python program MoverHonda12Final (listed below)
    - Python program MoverChopper21Final (listed below)
    - Python program MoverChopper22Final (listed below)
    - Python program MoverHonda21Final (listed below)
    - Python program MoverHonda22Final (listed below)
  - program Honda1Robot1 (3 instructions, listed below)
  - program Honda2Robot1 (3 instructions, listed below)
  - program Honda1Robot2 (3 instructions, listed below)
  - program Honda2Robot2 (3 instructions, listed below)
  - program Chopper1Robot1 (3 instructions, listed below)
  - program Chopper2Robot1 (3 instructions, listed below)
  - program Chopper1Robot2 (3 instructions, listed below)
  - program Chopper2Robot2 (3 instructions, listed below)

--- Python program Honda11 ---
from robodk.robolink import *  # API de RoboDK
from robodk.robomath import *  # Funciones matemáticas
import time
import math

# Inicializar conexión con RoboDK
RDK = Robolink()

# Borrar las partículas de pintura previas
RDK.Spray_Clear()

# Comprobar si estamos en modo simulación
if RDK.RunMode() != RUNMODE_SIMULATE:
    raise Exception('El robot no está en modo simulación')

# Obtener el robot
robot = RDK.Item('ABB IRB 580/12S 1', ITEM_TYPE_ROBOT)
if not robot.Valid():
    raise Exception('Robot "ABB IRB 580/12S 1" no encontrado')

# Establecer herramienta activa (TCP1)
tool = RDK.Item('TCP1', ITEM_TYPE_TOOL)
if not tool.Valid():
    raise Exception('Herramienta TCP1 no encontrada')
robot.setTool(tool)

# Obtener el objeto a pintar
honda = RDK.Item('Frame cb 750 1', ITEM_TYPE_OBJECT)
if not honda.Valid():
    raise Exception('Objeto "Frame cb 750 1" no encontrado')

# Obtener el sistema del gancho
frame6 = RDK.Item('Frame H1', ITEM_TYPE_FRAME)
if not frame6.Valid():
    raise Exception('Sistema "Frame H1" no encontrado')

# Obtener el sistema de la honda
frame5 = RDK.Item('Frame 5', ITEM_TYPE_FRAME)
if not frame5.Valid():
    raise Exception('Sistema "Frame 5" no encontrado')



# -------------------------
# MAPEO DE COLORES
# -------------------------
colores_numericos = {
    0: [1.0, 0.0, 0.0],  # rojo
    1: [0.0, 0.0, 0.0],  # negro
    2: [0.0, 1.0, 0.0],  # verde
    3: [0.5, 0.5, 0.5],  # gris
    4: [1.0, 1.0, 1.0],  # blanco
    5: [1.0, 0.5, 0.0]   # naranja
}

# Obtener número desde variable global de RoboDK
valor_color = RDK.getParam('ColorElegido1')
if valor_color is None:
    valor_color = 0  # valor por defecto
valor_color = int(valor_color)

if valor_color not in colores_numericos:
    raise Exception(f'ColorElegido inválido: {valor_color}')
color_final = colores_numericos[valor_color]

# Color neutro inicial
color_inicial = [0.9, 0.9, 0.9]

# Activar pintado automático
options_command = "ELLYPSE PROJECT PARTICLE=SPHERE(4,10,1,1,0.5) STEP=3x3 RAND=2"
close_param = [0, 0, 0, 5, 0, 0, 0, 5, 0, color_final[0], color_final[1], color_final[2], 1]
far_param   = [0, 0, 2000, 500, 0, 2000, 0, 500, 2000, color_final[0], color_final[1], color_final[2], 0.2]
volume = Mat([close_param, far_param]).tr()
RDK.Spray_Add(tool, honda, options_command, volume)
RDK.Spray_SetState(SPRAY_ON)

# Establecer velocidades lentas
robot.setSpeed(50, 50)
robot.setAcceleration(50)

# Lista de nombres de targets
targets = [
    'Pintura11_1',
    'Pintura12_1',
    'Pintura12_4',
    'Pintura12_3',
    'Pintura12_2',
    'Pintura12_5',
    'Pintura12_6',
    'Pintura12_7',
    'Pintura12_8',
    'Pintura12_9',
    'Pintura12_10',
    'Pintura12_9',
    'Pintura12_11',
    'Pintura12_9',
    'Pintura11_1',

    'Pintura12_13',
    'Pintura12_14',
    'Pintura12_15',
    'Pintura12_16',
    'Pintura12_17',
    'Pintura12_18',
    'Pintura12_19',
    'Pintura12_17',
    'Pintura12_16',
    'Pintura12_15',
    'Pintura12_23',
    'Pintura12_22',
    'Pintura12_24',
    'Pintura12_25',
    'Pintura12_13',
    'Pintura12_20',
    'Pintura12_21',
    'Pintura11_1',

    'Pintura12_26',
    'Pintura12_29',
    'Pintura12_28',
    'Pintura12_27',
    'Pintura12_30',
    'Pintura12_31',
    'Pintura12_32',
    'Pintura12_33',
    'Pintura12_34',
    'Pintura12_36',
    'Pintura12_35',
    'Pintura12_34',
    'Pintura12_26',
    'Pintura11_1',

    'Pintura12_37',
    'Pintura12_38',
    'Pintura12_39',
    'Pintura12_40',
    'Pintura12_41',
    'Pintura12_42',
    'Pintura12_43',
    'Pintura12_44',
    'Pintura12_45',
    'Pintura12_46',
    'Pintura12_47',
    'Pintura12_48',
    'Pintura12_49',
    'Pintura12_50',
    'Pintura11_1'


]

# Obtener poses de targets
target_poses = []

# Contar los pasos totales en todas las fases

step_index = 0

# Funcion para actualizar el color de la pieza
def actualizar_color(step_index, total_steps):
    factor = step_index / (total_steps - 1)
    rojo  = color_inicial[0] + (color_final[0] - color_inicial[0]) * factor
    verde = color_inicial[1] + (color_final[1] - color_inicial[1]) * factor
    azul  = color_inicial[2] + (color_final[2] - color_inicial[2]) * factor
    honda.setColor([rojo, verde, azul, 1.0])

for target_name in targets:
    target = RDK.Item(target_name, ITEM_TYPE_TARGET)
    if not target.Valid():
        raise Exception(f'Target no encontrado: {target_name}')
    target_poses.append(target.Pose())

total_steps = len(target_poses)

# Ir a posición de inicio
home_joints = robot.JointsHome()
robot.MoveJ(home_joints)
robot.MoveJ(target_poses[0])

RDK.Spray_SetState(SPRAY_ON)

# Pintado con cambio progresivo de color (10 pasos)
for i, pose in enumerate(target_poses[1:10]):

    actualizar_color(step_index, total_steps)
    robot.MoveL(pose)
    step_index += 1

# Últimos movimientos
robot.setSpeed(50, 50)
robot.setAcceleration(50)
actualizar_color(step_index, total_steps)
robot.MoveL(target_poses[10])
step_index += 1
actualizar_color(step_index, total_steps)
robot.MoveL(target_poses[11])
step_index += 1

robot.setSpeed(10, 10)
robot.setAcceleration(10)
for pose in target_poses[12:15]:
    actualizar_color(step_index, total_steps)
    robot.MoveJ(pose)
    step_index += 1

# Bucle: 18 pasos de 5 grados
for i in range(18):
    # Obtener la pose actual en cada iteración (actualizada)
    pose_actual6 = frame6.Pose()
    pose_actual5 = frame5.Pose()

    # Crear una rotación de 5 grados en Z
    rot_5deg6 = robomath.rotz(math.radians(5))
    rot_5deg5 = robomath.rotz(math.radians(5))

    # Aplicar rotación acumulativa
    nueva_pose6 = pose_actual6 * rot_5deg6
    nueva_pose5 = pose_actual5 * rot_5deg5

    # Establecer la nueva pose
    frame6.setPose(nueva_pose6)
    frame5.setPose(nueva_pose5)

for pose in target_poses[15:29]:
    actualizar_color(step_index, total_steps)
    robot.MoveJ(pose)
    step_index += 1

robot.MoveJ(home_joints)

for pose in target_poses[30:33]:
    actualizar_color(step_index, total_steps)
    robot.MoveJ(pose)
    step_index += 1

# Bucle: 18 pasos de 5 grados
for i in range(18):
    # Obtener la pose actual en cada iteración (actualizada)
    pose_actual6 = frame6.Pose()
    pose_actual5 = frame5.Pose()

    # Crear una rotación de 5 grados en Z
    rot_5deg6 = robomath.rotz(math.radians(5))
    rot_5deg5 = robomath.rotz(math.radians(5))

    # Aplicar rotación acumulativa
    nueva_pose6 = pose_actual6 * rot_5deg6
    nueva_pose5 = pose_actual5 * rot_5deg5

    # Establecer la nueva pose
    frame6.setPose(nueva_pose6)
    frame5.setPose(nueva_pose5)

for pose in target_poses[33:47]:
    actualizar_color(step_index, total_steps)
    robot.MoveJ(pose)
    step_index += 1

# Bucle: 18 pasos de 5 grados
for i in range(18):
    # Obtener la pose actual en cada iteración (actualizada)
    pose_actual6 = frame6.Pose()
    pose_actual5 = frame5.Pose()

    # Crear una rotación de 5 grados en Z
    rot_5deg6 = robomath.rotz(math.radians(5))
    rot_5deg5 = robomath.rotz(math.radians(5))

    # Aplicar rotación acumulativa
    nueva_pose6 = pose_actual6 * rot_5deg6
    nueva_pose5 = pose_actual5 * rot_5deg5

    # Establecer la nueva pose
    frame6.setPose(nueva_pose6)
    frame5.setPose(nueva_pose5)

for pose in target_poses[47:]:
    actualizar_color(step_index, total_steps)
    robot.MoveJ(pose)
    step_index += 1

# Bucle: 18 pasos de 5 grados
for i in range(18):
    # Obtener la pose actual en cada iteración (actualizada)
    pose_actual6 = frame6.Pose()
    pose_actual5 = frame5.Pose()

    # Crear una rotación de 5 grados en Z
    rot_5deg6 = robomath.rotz(math.radians(5))
    rot_5deg5 = robomath.rotz(math.radians(5))

    # Aplicar rotación acumulativa
    nueva_pose6 = pose_actual6 * rot_5deg6
    nueva_pose5 = pose_actual5 * rot_5deg5

    # Establecer la nueva pose
    frame6.setPose(nueva_pose6)
    frame5.setPose(nueva_pose5)

robot.MoveJ(home_joints)
time.sleep(5.0)

robot.MoveJ(home_joints)
robot.MoveJ(target_poses[0])

RDK.Spray_SetState(SPRAY_ON)

# Pintado con cambio progresivo de color (10 pasos)
for i, pose in enumerate(target_poses[1:10]):

    actualizar_color(step_index, total_steps)
    robot.MoveL(pose)
    step_index += 1

# Últimos movimientos
robot.setSpeed(50, 50)
robot.setAcceleration(50)
actualizar_color(step_index, total_steps)
robot.MoveL(target_poses[10])
step_index += 1
actualizar_color(step_index, total_steps)
robot.MoveL(target_poses[11])
step_index += 1

robot.setSpeed(10, 10)
robot.setAcceleration(10)
for pose in target_poses[12:15]:
    actualizar_color(step_index, total_steps)
    robot.MoveJ(pose)
    step_index += 1

# Bucle: 18 pasos de 5 grados
for i in range(18):
    # Obtener la pose actual en cada iteración (actualizada)
    pose_actual6 = frame6.Pose()
    pose_actual5 = frame5.Pose()

    # Crear una rotación de 5 grados en Z
    rot_5deg6 = robomath.rotz(math.radians(5))
    rot_5deg5 = robomath.rotz(math.radians(5))

    # Aplicar rotación acumulativa
    nueva_pose6 = pose_actual6 * rot_5deg6
    nueva_pose5 = pose_actual5 * rot_5deg5

    # Establecer la nueva pose
    frame6.setPose(nueva_pose6)
    frame5.setPose(nueva_pose5)

for pose in target_poses[15:29]:
    actualizar_color(step_index, total_steps)
    robot.MoveJ(pose)
    step_index += 1

robot.MoveJ(home_joints)

for pose in target_poses[30:33]:
    actualizar_color(step_index, total_steps)
    robot.MoveJ(pose)
    step_index += 1

# Bucle: 18 pasos de 5 grados
for i in range(18):
    # Obtener la pose actual en cada iteración (actualizada)
    pose_actual6 = frame6.Pose()
    pose_actual5 = frame5.Pose()

    # Crear una rotación de 5 grados en Z
    rot_5deg6 = robomath.rotz(math.radians(5))
    rot_5deg5 = robomath.rotz(math.radians(5))

    # Aplicar rotación acumulativa
    nueva_pose6 = pose_actual6 * rot_5deg6
    nueva_pose5 = pose_actual5 * rot_5deg5

    # Establecer la nueva pose
    frame6.setPose(nueva_pose6)
    frame5.setPose(nueva_pose5)

for pose in target_poses[33:47]:
    actualizar_color(step_index, total_steps)
    robot.MoveJ(pose)
    step_index += 1

# Bucle: 18 pasos de 5 grados
for i in range(18):
    # Obtener la pose actual en cada iteración (actualizada)
    pose_actual6 = frame6.Pose()
    pose_actual5 = frame5.Pose()

    # Crear una rotación de 5 grados en Z
    rot_5deg6 = robomath.rotz(math.radians(5))
    rot_5deg5 = robomath.rotz(math.radians(5))

    # Aplicar rotación acumulativa
    nueva_pose6 = pose_actual6 * rot_5deg6
    nueva_pose5 = pose_actual5 * rot_5deg5

    # Establecer la nueva pose
    frame6.setPose(nueva_pose6)
    frame5.setPose(nueva_pose5)

for pose in target_poses[47:]:
    actualizar_color(step_index, total_steps)
    robot.MoveJ(pose)
    step_index += 1

# Bucle: 18 pasos de 5 grados
for i in range(18):
    # Obtener la pose actual en cada iteración (actualizada)
    pose_actual6 = frame6.Pose()
    pose_actual5 = frame5.Pose()

    # Crear una rotación de 5 grados en Z
    rot_5deg6 = robomath.rotz(math.radians(5))
    rot_5deg5 = robomath.rotz(math.radians(5))

    # Aplicar rotación acumulativa
    nueva_pose6 = pose_actual6 * rot_5deg6
    nueva_pose5 = pose_actual5 * rot_5deg5

    # Establecer la nueva pose
    frame6.setPose(nueva_pose6)
    frame5.setPose(nueva_pose5)

# Desactivar pintado al finalizar
RDK.Spray_Clear()
RDK.Spray_SetState(SPRAY_OFF)

--- Python program Honda12 ---
from robodk.robolink import *  # API de RoboDK
from robodk.robomath import *  # Funciones matemáticas
import time
import math

# Inicializar conexión con RoboDK
RDK = Robolink()

# Borrar las partículas de pintura previas
RDK.Spray_Clear()

# Comprobar si estamos en modo simulación
if RDK.RunMode() != RUNMODE_SIMULATE:
    raise Exception('El robot no está en modo simulación')

# Obtener el robot
robot = RDK.Item('ABB IRB 580/12S 1', ITEM_TYPE_ROBOT)
if not robot.Valid():
    raise Exception('Robot "ABB IRB 580/12S 1" no encontrado')

# Establecer herramienta activa (TCP1)
tool = RDK.Item('TCP1', ITEM_TYPE_TOOL)
if not tool.Valid():
    raise Exception('Herramienta TCP1 no encontrada')
robot.setTool(tool)

# Obtener el objeto a pintar
honda = RDK.Item('Frame cb 750 2', ITEM_TYPE_OBJECT)
if not honda.Valid():
    raise Exception('Objeto "Frame cb 750 2" no encontrado')

# Obtener el sistema del gancho
frame6 = RDK.Item('Frame H2', ITEM_TYPE_FRAME)
if not frame6.Valid():
    raise Exception('Sistema "Frame H2" no encontrado')

# Obtener el sistema de la honda
frame5 = RDK.Item('Frame 7', ITEM_TYPE_FRAME)
if not frame5.Valid():
    raise Exception('Sistema "Frame 7" no encontrado')



# -------------------------
# MAPEO DE COLORES
# -------------------------
colores_numericos = {
    0: [1.0, 0.0, 0.0],  # rojo
    1: [0.0, 0.0, 0.0],  # negro
    2: [0.0, 1.0, 0.0],  # verde
    3: [0.5, 0.5, 0.5],  # gris
    4: [1.0, 1.0, 1.0],  # blanco
    5: [1.0, 0.5, 0.0]   # naranja
}

# Obtener número desde variable global de RoboDK
valor_color = RDK.getParam('ColorElegido1')
if valor_color is None:
    valor_color = 0  # valor por defecto
valor_color = int(valor_color)

if valor_color not in colores_numericos:
    raise Exception(f'ColorElegido inválido: {valor_color}')
color_final = colores_numericos[valor_color]

# Color neutro inicial
color_inicial = [0.9, 0.9, 0.9]

# Activar pintado automático
options_command = "ELLYPSE PROJECT PARTICLE=SPHERE(4,10,1,1,0.5) STEP=3x3 RAND=2"
close_param = [0, 0, 0, 5, 0, 0, 0, 5, 0, color_final[0], color_final[1], color_final[2], 1]
far_param   = [0, 0, 2000, 500, 0, 2000, 0, 500, 2000, color_final[0], color_final[1], color_final[2], 0.2]
volume = Mat([close_param, far_param]).tr()
RDK.Spray_Add(tool, honda, options_command, volume)
RDK.Spray_SetState(SPRAY_ON)

# Establecer velocidades lentas
robot.setSpeed(50, 50)
robot.setAcceleration(50)

# Lista de nombres de targets
targets = [
    'Pintura11_1',
    'Pintura12_1',
    'Pintura12_4',
    'Pintura12_3',
    'Pintura12_2',
    'Pintura12_5',
    'Pintura12_6',
    'Pintura12_7',
    'Pintura12_8',
    'Pintura12_9',
    'Pintura12_10',
    'Pintura12_9',
    'Pintura12_11',
    'Pintura12_9',
    'Pintura11_1',

    'Pintura12_13',
    'Pintura12_14',
    'Pintura12_15',
    'Pintura12_16',
    'Pintura12_17',
    'Pintura12_18',
    'Pintura12_19',
    'Pintura12_17',
    'Pintura12_16',
    'Pintura12_15',
    'Pintura12_23',
    'Pintura12_22',
    'Pintura12_24',
    'Pintura12_25',
    'Pintura12_13',
    'Pintura12_20',
    'Pintura12_21',
    'Pintura11_1',

    'Pintura12_26',
    'Pintura12_29',
    'Pintura12_28',
    'Pintura12_27',
    'Pintura12_30',
    'Pintura12_31',
    'Pintura12_32',
    'Pintura12_33',
    'Pintura12_34',
    'Pintura12_36',
    'Pintura12_35',
    'Pintura12_34',
    'Pintura12_26',
    'Pintura11_1',

    'Pintura12_37',
    'Pintura12_38',
    'Pintura12_39',
    'Pintura12_40',
    'Pintura12_41',
    'Pintura12_42',
    'Pintura12_43',
    'Pintura12_44',
    'Pintura12_45',
    'Pintura12_46',
    'Pintura12_47',
    'Pintura12_48',
    'Pintura12_49',
    'Pintura12_50',
    'Pintura11_1'


]

# Obtener poses de targets
target_poses = []

# Contar los pasos totales en todas las fases

step_index = 0

# Funcion para actualizar el color de la pieza
def actualizar_color(step_index, total_steps):
    factor = step_index / (total_steps - 1)
    rojo  = color_inicial[0] + (color_final[0] - color_inicial[0]) * factor
    verde = color_inicial[1] + (color_final[1] - color_inicial[1]) * factor
    azul  = color_inicial[2] + (color_final[2] - color_inicial[2]) * factor
    honda.setColor([rojo, verde, azul, 1.0])

for target_name in targets:
    target = RDK.Item(target_name, ITEM_TYPE_TARGET)
    if not target.Valid():
        raise Exception(f'Target no encontrado: {target_name}')
    target_poses.append(target.Pose())

total_steps = len(target_poses)

# Ir a posición de inicio
home_joints = robot.JointsHome()
robot.MoveJ(home_joints)
robot.MoveJ(target_poses[0])

RDK.Spray_SetState(SPRAY_ON)

# Pintado con cambio progresivo de color (10 pasos)
for i, pose in enumerate(target_poses[1:10]):

    actualizar_color(step_index, total_steps)
    robot.MoveL(pose)
    step_index += 1

# Últimos movimientos
robot.setSpeed(50, 50)
robot.setAcceleration(50)
actualizar_color(step_index, total_steps)
robot.MoveL(target_poses[10])
step_index += 1
actualizar_color(step_index, total_steps)
robot.MoveL(target_poses[11])
step_index += 1

robot.setSpeed(10, 10)
robot.setAcceleration(10)
for pose in target_poses[12:15]:
    actualizar_color(step_index, total_steps)
    robot.MoveJ(pose)
    step_index += 1

# Bucle: 18 pasos de 5 grados
for i in range(18):
    # Obtener la pose actual en cada iteración (actualizada)
    pose_actual6 = frame6.Pose()
    pose_actual5 = frame5.Pose()

    # Crear una rotación de 5 grados en Z
    rot_5deg6 = robomath.rotz(math.radians(5))
    rot_5deg5 = robomath.rotz(math.radians(5))

    # Aplicar rotación acumulativa
    nueva_pose6 = pose_actual6 * rot_5deg6
    nueva_pose5 = pose_actual5 * rot_5deg5

    # Establecer la nueva pose
    frame6.setPose(nueva_pose6)
    frame5.setPose(nueva_pose5)

for pose in target_poses[15:29]:
    actualizar_color(step_index, total_steps)
    robot.MoveJ(pose)
    step_index += 1

robot.MoveJ(home_joints)

for pose in target_poses[30:33]:
    actualizar_color(step_index, total_steps)
    robot.MoveJ(pose)
    step_index += 1

# Bucle: 18 pasos de 5 grados
for i in range(18):
    # Obtener la pose actual en cada iteración (actualizada)
    pose_actual6 = frame6.Pose()
    pose_actual5 = frame5.Pose()

    # Crear una rotación de 5 grados en Z
    rot_5deg6 = robomath.rotz(math.radians(5))
    rot_5deg5 = robomath.rotz(math.radians(5))

    # Aplicar rotación acumulativa
    nueva_pose6 = pose_actual6 * rot_5deg6
    nueva_pose5 = pose_actual5 * rot_5deg5

    # Establecer la nueva pose
    frame6.setPose(nueva_pose6)
    frame5.setPose(nueva_pose5)

for pose in target_poses[33:47]:
    actualizar_color(step_index, total_steps)
    robot.MoveJ(pose)
    step_index += 1

# Bucle: 18 pasos de 5 grados
for i in range(18):
    # Obtener la pose actual en cada iteración (actualizada)
    pose_actual6 = frame6.Pose()
    pose_actual5 = frame5.Pose()

    # Crear una rotación de 5 grados en Z
    rot_5deg6 = robomath.rotz(math.radians(5))
    rot_5deg5 = robomath.rotz(math.radians(5))

    # Aplicar rotación acumulativa
    nueva_pose6 = pose_actual6 * rot_5deg6
    nueva_pose5 = pose_actual5 * rot_5deg5

    # Establecer la nueva pose
    frame6.setPose(nueva_pose6)
    frame5.setPose(nueva_pose5)

for pose in target_poses[47:]:
    actualizar_color(step_index, total_steps)
    robot.MoveJ(pose)
    step_index += 1

# Bucle: 18 pasos de 5 grados
for i in range(18):
    # Obtener la pose actual en cada iteración (actualizada)
    pose_actual6 = frame6.Pose()
    pose_actual5 = frame5.Pose()

    # Crear una rotación de 5 grados en Z
    rot_5deg6 = robomath.rotz(math.radians(5))
    rot_5deg5 = robomath.rotz(math.radians(5))

    # Aplicar rotación acumulativa
    nueva_pose6 = pose_actual6 * rot_5deg6
    nueva_pose5 = pose_actual5 * rot_5deg5

    # Establecer la nueva pose
    frame6.setPose(nueva_pose6)
    frame5.setPose(nueva_pose5)

robot.MoveJ(home_joints)
time.sleep(5.0)

robot.MoveJ(home_joints)
robot.MoveJ(target_poses[0])

RDK.Spray_SetState(SPRAY_ON)

# Pintado con cambio progresivo de color (10 pasos)
for i, pose in enumerate(target_poses[1:10]):

    actualizar_color(step_index, total_steps)
    robot.MoveL(pose)
    step_index += 1

# Últimos movimientos
robot.setSpeed(50, 50)
robot.setAcceleration(50)
actualizar_color(step_index, total_steps)
robot.MoveL(target_poses[10])
step_index += 1
actualizar_color(step_index, total_steps)
robot.MoveL(target_poses[11])
step_index += 1

robot.setSpeed(10, 10)
robot.setAcceleration(10)
for pose in target_poses[12:15]:
    actualizar_color(step_index, total_steps)
    robot.MoveJ(pose)
    step_index += 1

# Bucle: 18 pasos de 5 grados
for i in range(18):
    # Obtener la pose actual en cada iteración (actualizada)
    pose_actual6 = frame6.Pose()
    pose_actual5 = frame5.Pose()

    # Crear una rotación de 5 grados en Z
    rot_5deg6 = robomath.rotz(math.radians(5))
    rot_5deg5 = robomath.rotz(math.radians(5))

    # Aplicar rotación acumulativa
    nueva_pose6 = pose_actual6 * rot_5deg6
    nueva_pose5 = pose_actual5 * rot_5deg5

    # Establecer la nueva pose
    frame6.setPose(nueva_pose6)
    frame5.setPose(nueva_pose5)

for pose in target_poses[15:29]:
    actualizar_color(step_index, total_steps)
    robot.MoveJ(pose)
    step_index += 1

robot.MoveJ(home_joints)

for pose in target_poses[30:33]:
    actualizar_color(step_index, total_steps)
    robot.MoveJ(pose)
    step_index += 1

# Bucle: 18 pasos de 5 grados
for i in range(18):
    # Obtener la pose actual en cada iteración (actualizada)
    pose_actual6 = frame6.Pose()
    pose_actual5 = frame5.Pose()

    # Crear una rotación de 5 grados en Z
    rot_5deg6 = robomath.rotz(math.radians(5))
    rot_5deg5 = robomath.rotz(math.radians(5))

    # Aplicar rotación acumulativa
    nueva_pose6 = pose_actual6 * rot_5deg6
    nueva_pose5 = pose_actual5 * rot_5deg5

    # Establecer la nueva pose
    frame6.setPose(nueva_pose6)
    frame5.setPose(nueva_pose5)

for pose in target_poses[33:47]:
    actualizar_color(step_index, total_steps)
    robot.MoveJ(pose)
    step_index += 1

# Bucle: 18 pasos de 5 grados
for i in range(18):
    # Obtener la pose actual en cada iteración (actualizada)
    pose_actual6 = frame6.Pose()
    pose_actual5 = frame5.Pose()

    # Crear una rotación de 5 grados en Z
    rot_5deg6 = robomath.rotz(math.radians(5))
    rot_5deg5 = robomath.rotz(math.radians(5))

    # Aplicar rotación acumulativa
    nueva_pose6 = pose_actual6 * rot_5deg6
    nueva_pose5 = pose_actual5 * rot_5deg5

    # Establecer la nueva pose
    frame6.setPose(nueva_pose6)
    frame5.setPose(nueva_pose5)

for pose in target_poses[47:]:
    actualizar_color(step_index, total_steps)
    robot.MoveJ(pose)
    step_index += 1

# Bucle: 18 pasos de 5 grados
for i in range(18):
    # Obtener la pose actual en cada iteración (actualizada)
    pose_actual6 = frame6.Pose()
    pose_actual5 = frame5.Pose()

    # Crear una rotación de 5 grados en Z
    rot_5deg6 = robomath.rotz(math.radians(5))
    rot_5deg5 = robomath.rotz(math.radians(5))

    # Aplicar rotación acumulativa
    nueva_pose6 = pose_actual6 * rot_5deg6
    nueva_pose5 = pose_actual5 * rot_5deg5

    # Establecer la nueva pose
    frame6.setPose(nueva_pose6)
    frame5.setPose(nueva_pose5)

# Desactivar pintado al finalizar
RDK.Spray_Clear()
RDK.Spray_SetState(SPRAY_OFF)

--- Python program Chopper11 ---
from robodk.robolink import *  # API de RoboDK
from robodk.robomath import *  # Funciones matemáticas
import time
import math

# Inicializar conexión con RoboDK
RDK = Robolink()

# Borrar las partículas de pintura previas
RDK.Spray_Clear()

# Comprobar si estamos en modo simulación
if RDK.RunMode() != RUNMODE_SIMULATE:
    raise Exception('El robot no está en modo simulación')

# Obtener el robot
robot = RDK.Item('ABB IRB 580/12S 1', ITEM_TYPE_ROBOT)
if not robot.Valid():
    raise Exception('Robot "ABB IRB 580/12S 1" no encontrado')

# Establecer herramienta activa (TCP1)
tool = RDK.Item('TCP1', ITEM_TYPE_TOOL)
if not tool.Valid():
    raise Exception('Herramienta TCP1 no encontrada')
robot.setTool(tool)

# Obtener el objeto a pintar
obj = RDK.Item('Chopper Frame AP203 1', ITEM_TYPE_OBJECT)
if not obj.Valid():
    raise Exception('Objeto "Chopper Frame AP203 1" no encontrado')

# Obtener el sistema del gancho
frame6 = RDK.Item('Frame C1', ITEM_TYPE_FRAME)
if not frame6.Valid():
    raise Exception('Sistema "Frame C1" no encontrado')

# Obtener el sistema del objeto
frame4 = RDK.Item('Frame 4', ITEM_TYPE_FRAME)
if not frame4.Valid():
    raise Exception('Sistema "Frame 4" no encontrado')

# -------------------------
# MAPEO DE COLORES
# -------------------------
colores_numericos = {
    0: [1.0, 0.0, 0.0],  # rojo
    1: [0.0, 0.0, 0.0],  # negro
    2: [0.0, 1.0, 0.0],  # verde
    3: [0.5, 0.5, 0.5],  # gris
    4: [1.0, 1.0, 1.0],  # blanco
    5: [1.0, 0.5, 0.0]   # naranja
}

# Obtener número desde variable global de RoboDK
valor_color = RDK.getParam('ColorElegido1')
if valor_color is None:
    valor_color = 0  # valor por defecto
valor_color = int(valor_color)

if valor_color not in colores_numericos:
    raise Exception(f'ColorElegido inválido: {valor_color}')
color_final = colores_numericos[valor_color]

# Color neutro inicial
color_inicial = [0.9, 0.9, 0.9]

# Activar pintado automático
options_command = f"ELLYPSE PROJECT PARTICLE=SPHERE(4,10,1,1,0.5) STEP=3x3 RAND=2"
close_param = [0, 0, 0, 5, 0, 0, 0, 5, 0, color_final[0], color_final[1], color_final[2], 1]
far_param   = [0, 0, 2000, 500, 0, 2000, 0, 500, 2000, color_final[0], color_final[1], color_final[2], 0.2]
volume = Mat([close_param, far_param]).tr()
RDK.Spray_Add(tool, obj, options_command, volume)
RDK.Spray_SetState(SPRAY_ON)

# Establecer velocidades lentas
robot.setSpeed(50, 50)
robot.setAcceleration(50)

# Lista de nombres de targets
targets = [
    'Pintura11_1',
    'Pintura11_2',
    'Pintura11_3',
    'Pintura11_4',
    'Pintura11_5',
    'Pintura11_6',
    'Pintura11_7',
    'Pintura11_8',
    'Pintura11_9',
    'Pintura11_8',
    'Pintura11_1',

    'Pintura11_11',
    'Pintura11_13',
    'Pintura11_14',
    'Pintura11_15',
    'Pintura11_16',
    'Pintura11_17',
    'Pintura11_18',
    'Pintura11_19',
    'Pintura11_13',
    'Pintura11_20',
    'Pintura11_1',

    'Pintura11_21',
    'Pintura11_22',
    'Pintura11_23',
    'Pintura11_24',
    'Pintura11_25',
    'Pintura11_26',
    'Pintura11_27',
    'Pintura11_28',
    'Pintura11_29',
    'Pintura11_28',
    'Pintura11_1',

    'Pintura11_31',
    'Pintura11_32',
    'Pintura11_39',
    'Pintura11_32',
    'Pintura11_33',
    'Pintura11_38',
    'Pintura11_34',
    'Pintura11_37',
    'Pintura11_35',
    'Pintura11_36',
    'Pintura11_37',
    'Pintura11_38',
    'Pintura11_39',
    'Pintura11_40'


]

# Obtener poses de targets
target_poses = []

# Contar los pasos totales en todas las fases

step_index = 0

# Funcion para actualizar el color de la pieza
def actualizar_color(step_index, total_steps):
    factor = step_index / (total_steps - 1)
    rojo  = color_inicial[0] + (color_final[0] - color_inicial[0]) * factor
    verde = color_inicial[1] + (color_final[1] - color_inicial[1]) * factor
    azul  = color_inicial[2] + (color_final[2] - color_inicial[2]) * factor
    obj.setColor([rojo, verde, azul, 1.0])

# Obtener poses desde los nombres de target
for target_name in targets:
    target = RDK.Item(target_name, ITEM_TYPE_TARGET)
    if not target.Valid():
        raise Exception(f'Target no encontrado: {target_name}')
    target_poses.append(target.Pose())

total_steps = len(target_poses)

# Ir a posición de inicio
home_joints = robot.JointsHome()
robot.MoveJ(home_joints)
robot.MoveJ(target_poses[0])

RDK.Spray_SetState(SPRAY_ON)

robot.setSpeed(10, 10)
robot.setAcceleration(10)

# Pintado con cambio progresivo de color (10 pasos)
for i, pose in enumerate(target_poses[1:10]):

    actualizar_color(step_index, total_steps)
    robot.MoveJ(pose)
    step_index += 1

# Últimos movimientos

robot.setSpeed(50, 50)
robot.setAcceleration(50)

actualizar_color(step_index, total_steps)
robot.MoveL(target_poses[11])
step_index += 1

# Bucle: 18 pasos de 5 grados
for i in range(18):
    # Obtener la pose actual en cada iteración (actualizada)
    pose_actual6 = frame6.Pose()
    pose_actual5 = frame4.Pose()

    # Crear una rotación de 5 grados en Z
    rot_5deg6 = robomath.rotz(math.radians(5))
    rot_5deg5 = robomath.rotz(math.radians(5))

    # Aplicar rotación acumulativa
    nueva_pose6 = pose_actual6 * rot_5deg6
    nueva_pose5 = pose_actual5 * rot_5deg5

    # Establecer la nueva pose
    frame6.setPose(nueva_pose6)
    frame4.setPose(nueva_pose5)

robot.setSpeed(10, 10)
robot.setAcceleration(10)

for pose in target_poses[12:23]:
    actualizar_color(step_index, total_steps)
    robot.MoveJ(pose)
    step_index += 1

# Bucle: 18 pasos de 5 grados
for i in range(18):
    # Obtener la pose actual en cada iteración (actualizada)
    pose_actual6 = frame6.Pose()
    pose_actual5 = frame4.Pose()

    # Crear una rotación de 5 grados en Z
    rot_5deg6 = robomath.rotz(math.radians(5))
    rot_5deg5 = robomath.rotz(math.radians(5))

    # Aplicar rotación acumulativa
    nueva_pose6 = pose_actual6 * rot_5deg6
    nueva_pose5 = pose_actual5 * rot_5deg5

    # Establecer la nueva pose
    frame6.setPose(nueva_pose6)
    frame4.setPose(nueva_pose5)

for pose in target_poses[23:33]:
    actualizar_color(step_index, total_steps)
    robot.MoveJ(pose)
    step_index += 1

robot.MoveJ(home_joints)

# Bucle: 18 pasos de 5 grados
for i in range(18):
    # Obtener la pose actual en cada iteración (actualizada)
    pose_actual6 = frame6.Pose()
    pose_actual5 = frame4.Pose()

    # Crear una rotación de 5 grados en Z
    rot_5deg6 = robomath.rotz(math.radians(5))
    rot_5deg5 = robomath.rotz(math.radians(5))

    # Aplicar rotación acumulativa
    nueva_pose6 = pose_actual6 * rot_5deg6
    nueva_pose5 = pose_actual5 * rot_5deg5

    # Establecer la nueva pose
    frame6.setPose(nueva_pose6)
    frame4.setPose(nueva_pose5)

for pose in target_poses[33:]:
    actualizar_color(step_index, total_steps)
    robot.MoveJ(pose)
    step_index += 1

robot.MoveJ(home_joints)

# Bucle: 18 pasos de 5 grados
for i in range(18):
    # Obtener la pose actual en cada iteración (actualizada)
    pose_actual6 = frame6.Pose()
    pose_actual5 = frame4.Pose()

    # Crear una rotación de 5 grados en Z
    rot_5deg6 = robomath.rotz(math.radians(5))
    rot_5deg5 = robomath.rotz(math.radians(5))

    # Aplicar rotación acumulativa
    nueva_pose6 = pose_actual6 * rot_5deg6
    nueva_pose5 = pose_actual5 * rot_5deg5

    # Establecer la nueva pose
    frame6.setPose(nueva_pose6)
    frame4.setPose(nueva_pose5)

robot.MoveJ(home_joints)
time.sleep(5.0)

robot.MoveJ(home_joints)
robot.MoveJ(target_poses[0])

RDK.Spray_SetState(SPRAY_ON)

robot.setSpeed(10, 10)
robot.setAcceleration(10)

# Pintado con cambio progresivo de color (10 pasos)
for i, pose in enumerate(target_poses[1:10]):

    actualizar_color(step_index, total_steps)
    robot.MoveJ(pose)
    step_index += 1

# Últimos movimientos

robot.setSpeed(50, 50)
robot.setAcceleration(50)

actualizar_color(step_index, total_steps)
robot.MoveL(target_poses[11])
step_index += 1

# Bucle: 18 pasos de 5 grados
for i in range(18):
    # Obtener la pose actual en cada iteración (actualizada)
    pose_actual6 = frame6.Pose()
    pose_actual5 = frame4.Pose()

    # Crear una rotación de 5 grados en Z
    rot_5deg6 = robomath.rotz(math.radians(5))
    rot_5deg5 = robomath.rotz(math.radians(5))

    # Aplicar rotación acumulativa
    nueva_pose6 = pose_actual6 * rot_5deg6
    nueva_pose5 = pose_actual5 * rot_5deg5

    # Establecer la nueva pose
    frame6.setPose(nueva_pose6)
    frame4.setPose(nueva_pose5)

robot.setSpeed(10, 10)
robot.setAcceleration(10)

for pose in target_poses[12:23]:
    actualizar_color(step_index, total_steps)
    robot.MoveJ(pose)
    step_index += 1

# Bucle: 18 pasos de 5 grados
for i in range(18):
    # Obtener la pose actual en cada iteración (actualizada)
    pose_actual6 = frame6.Pose()
    pose_actual5 = frame4.Pose()

    # Crear una rotación de 5 grados en Z
    rot_5deg6 = robomath.rotz(math.radians(5))
    rot_5deg5 = robomath.rotz(math.radians(5))

    # Aplicar rotación acumulativa
    nueva_pose6 = pose_actual6 * rot_5deg6
    nueva_pose5 = pose_actual5 * rot_5deg5

    # Establecer la nueva pose
    frame6.setPose(nueva_pose6)
    frame4.setPose(nueva_pose5)

for pose in target_poses[23:33]:
    actualizar_color(step_index, total_steps)
    robot.MoveJ(pose)
    step_index += 1

robot.MoveJ(home_joints)

# Bucle: 18 pasos de 5 grados
for i in range(18):
    # Obtener la pose actual en cada iteración (actualizada)
    pose_actual6 = frame6.Pose()
    pose_actual5 = frame4.Pose()

    # Crear una rotación de 5 grados en Z
    rot_5deg6 = robomath.rotz(math.radians(5))
    rot_5deg5 = robomath.rotz(math.radians(5))

    # Aplicar rotación acumulativa
    nueva_pose6 = pose_actual6 * rot_5deg6
    nueva_pose5 = pose_actual5 * rot_5deg5

    # Establecer la nueva pose
    frame6.setPose(nueva_pose6)
    frame4.setPose(nueva_pose5)

for pose in target_poses[33:]:
    actualizar_color(step_index, total_steps)
    robot.MoveJ(pose)
    step_index += 1

robot.MoveJ(home_joints)

# Bucle: 18 pasos de 5 grados
for i in range(18):
    # Obtener la pose actual en cada iteración (actualizada)
    pose_actual6 = frame6.Pose()
    pose_actual5 = frame4.Pose()

    # Crear una rotación de 5 grados en Z
    rot_5deg6 = robomath.rotz(math.radians(5))
    rot_5deg5 = robomath.rotz(math.radians(5))

    # Aplicar rotación acumulativa
    nueva_pose6 = pose_actual6 * rot_5deg6
    nueva_pose5 = pose_actual5 * rot_5deg5

    # Establecer la nueva pose
    frame6.setPose(nueva_pose6)
    frame4.setPose(nueva_pose5)

# Desactivar pintado al finalizar
RDK.Spray_Clear()
RDK.Spray_SetState(SPRAY_OFF)

--- Python program Chopper12 ---
from robodk.robolink import *  # API de RoboDK
from robodk.robomath import *  # Funciones matemáticas
import time
import math

# Inicializar conexión con RoboDK
RDK = Robolink()

# Borrar las partículas de pintura previas
RDK.Spray_Clear()

# Comprobar si estamos en modo simulación
if RDK.RunMode() != RUNMODE_SIMULATE:
    raise Exception('El robot no está en modo simulación')

# Obtener el robot
robot = RDK.Item('ABB IRB 580/12S 1', ITEM_TYPE_ROBOT)
if not robot.Valid():
    raise Exception('Robot "ABB IRB 580/12S 1" no encontrado')

# Establecer herramienta activa (TCP1)
tool = RDK.Item('TCP1', ITEM_TYPE_TOOL)
if not tool.Valid():
    raise Exception('Herramienta TCP1 no encontrada')
robot.setTool(tool)

# Obtener el objeto a pintar
obj = RDK.Item('Chopper Frame AP203 2', ITEM_TYPE_OBJECT)
if not obj.Valid():
    raise Exception('Objeto "Chopper Frame AP203 2" no encontrado')

# Obtener el sistema del gancho
frame6 = RDK.Item('Frame C2', ITEM_TYPE_FRAME)
if not frame6.Valid():
    raise Exception('Sistema "Frame C2" no encontrado')

# Obtener el sistema del objeto
frame4 = RDK.Item('Frame 6', ITEM_TYPE_FRAME)
if not frame4.Valid():
    raise Exception('Sistema "Frame 6" no encontrado')

# -------------------------
# MAPEO DE COLORES
# -------------------------
colores_numericos = {
    0: [1.0, 0.0, 0.0],  # rojo
    1: [0.0, 0.0, 0.0],  # negro
    2: [0.0, 1.0, 0.0],  # verde
    3: [0.5, 0.5, 0.5],  # gris
    4: [1.0, 1.0, 1.0],  # blanco
    5: [1.0, 0.5, 0.0]   # naranja
}

# Obtener número desde variable global de RoboDK
valor_color = RDK.getParam('ColorElegido1')
if valor_color is None:
    valor_color = 0  # valor por defecto
valor_color = int(valor_color)

if valor_color not in colores_numericos:
    raise Exception(f'ColorElegido inválido: {valor_color}')
color_final = colores_numericos[valor_color]

# Color neutro inicial
color_inicial = [0.9, 0.9, 0.9]

# Activar pintado automático
options_command = f"ELLYPSE PROJECT PARTICLE=SPHERE(4,10,1,1,0.5) STEP=3x3 RAND=2"
close_param = [0, 0, 0, 5, 0, 0, 0, 5, 0, color_final[0], color_final[1], color_final[2], 1]
far_param   = [0, 0, 2000, 500, 0, 2000, 0, 500, 2000, color_final[0], color_final[1], color_final[2], 0.2]
volume = Mat([close_param, far_param]).tr()
RDK.Spray_Add(tool, obj, options_command, volume)
RDK.Spray_SetState(SPRAY_ON)

# Establecer velocidades lentas
robot.setSpeed(50, 50)
robot.setAcceleration(50)

# Lista de nombres de targets
targets = [
    'Pintura11_1',
    'Pintura11_2',
    'Pintura11_3',
    'Pintura11_4',
    'Pintura11_5',
    'Pintura11_6',
    'Pintura11_7',
    'Pintura11_8',
    'Pintura11_9',
    'Pintura11_8',
    'Pintura11_1',

    'Pintura11_11',
    'Pintura11_13',
    'Pintura11_14',
    'Pintura11_15',
    'Pintura11_16',
    'Pintura11_17',
    'Pintura11_18',
    'Pintura11_19',
    'Pintura11_13',
    'Pintura11_20',
    'Pintura11_1',

    'Pintura11_21',
    'Pintura11_22',
    'Pintura11_23',
    'Pintura11_24',
    'Pintura11_25',
    'Pintura11_26',
    'Pintura11_27',
    'Pintura11_28',
    'Pintura11_29',
    'Pintura11_28',
    'Pintura11_1',

    'Pintura11_31',
    'Pintura11_32',
    'Pintura11_39',
    'Pintura11_32',
    'Pintura11_33',
    'Pintura11_38',
    'Pintura11_34',
    'Pintura11_37',
    'Pintura11_35',
    'Pintura11_36',
    'Pintura11_37',
    'Pintura11_38',
    'Pintura11_39',
    'Pintura11_40'


]

# Obtener poses de targets
target_poses = []

# Contar los pasos totales en todas las fases

step_index = 0

# Funcion para actualizar el color de la pieza
def actualizar_color(step_index, total_steps):
    factor = step_index / (total_steps - 1)
    rojo  = color_inicial[0] + (color_final[0] - color_inicial[0]) * factor
    verde = color_inicial[1] + (color_final[1] - color_inicial[1]) * factor
    azul  = color_inicial[2] + (color_final[2] - color_inicial[2]) * factor
    obj.setColor([rojo, verde, azul, 1.0])

# Obtener poses desde los nombres de target
for target_name in targets:
    target = RDK.Item(target_name, ITEM_TYPE_TARGET)
    if not target.Valid():
        raise Exception(f'Target no encontrado: {target_name}')
    target_poses.append(target.Pose())

total_steps = len(target_poses)

# Ir a posición de inicio
home_joints = robot.JointsHome()
robot.MoveJ(home_joints)
robot.MoveJ(target_poses[0])

RDK.Spray_SetState(SPRAY_ON)

robot.setSpeed(10, 10)
robot.setAcceleration(10)

# Pintado con cambio progresivo de color (10 pasos)
for i, pose in enumerate(target_poses[1:10]):

    actualizar_color(step_index, total_steps)
    robot.MoveJ(pose)
    step_index += 1

# Últimos movimientos

robot.setSpeed(50, 50)
robot.setAcceleration(50)

actualizar_color(step_index, total_steps)
robot.MoveL(target_poses[11])
step_index += 1

# Bucle: 18 pasos de 5 grados
for i in range(18):
    # Obtener la pose actual en cada iteración (actualizada)
    pose_actual6 = frame6.Pose()
    pose_actual5 = frame4.Pose()

    # Crear una rotación de 5 grados en Z
    rot_5deg6 = robomath.rotz(math.radians(5))
    rot_5deg5 = robomath.rotz(math.radians(5))

    # Aplicar rotación acumulativa
    nueva_pose6 = pose_actual6 * rot_5deg6
    nueva_pose5 = pose_actual5 * rot_5deg5

    # Establecer la nueva pose
    frame6.setPose(nueva_pose6)
    frame4.setPose(nueva_pose5)

robot.setSpeed(10, 10)
robot.setAcceleration(10)

for pose in target_poses[12:23]:
    actualizar_color(step_index, total_steps)
    robot.MoveJ(pose)
    step_index += 1

# Bucle: 18 pasos de 5 grados
for i in range(18):
    # Obtener la pose actual en cada iteración (actualizada)
    pose_actual6 = frame6.Pose()
    pose_actual5 = frame4.Pose()

    # Crear una rotación de 5 grados en Z
    rot_5deg6 = robomath.rotz(math.radians(5))
    rot_5deg5 = robomath.rotz(math.radians(5))

    # Aplicar rotación acumulativa
    nueva_pose6 = pose_actual6 * rot_5deg6
    nueva_pose5 = pose_actual5 * rot_5deg5

    # Establecer la nueva pose
    frame6.setPose(nueva_pose6)
    frame4.setPose(nueva_pose5)

for pose in target_poses[23:33]:
    actualizar_color(step_index, total_steps)
    robot.MoveJ(pose)
    step_index += 1

robot.MoveJ(home_joints)

# Bucle: 18 pasos de 5 grados
for i in range(18):
    # Obtener la pose actual en cada iteración (actualizada)
    pose_actual6 = frame6.Pose()
    pose_actual5 = frame4.Pose()

    # Crear una rotación de 5 grados en Z
    rot_5deg6 = robomath.rotz(math.radians(5))
    rot_5deg5 = robomath.rotz(math.radians(5))

    # Aplicar rotación acumulativa
    nueva_pose6 = pose_actual6 * rot_5deg6
    nueva_pose5 = pose_actual5 * rot_5deg5

    # Establecer la nueva pose
    frame6.setPose(nueva_pose6)
    frame4.setPose(nueva_pose5)

for pose in target_poses[33:]:
    actualizar_color(step_index, total_steps)
    robot.MoveJ(pose)
    step_index += 1

robot.MoveJ(home_joints)

# Bucle: 18 pasos de 5 grados
for i in range(18):
    # Obtener la pose actual en cada iteración (actualizada)
    pose_actual6 = frame6.Pose()
    pose_actual5 = frame4.Pose()

    # Crear una rotación de 5 grados en Z
    rot_5deg6 = robomath.rotz(math.radians(5))
    rot_5deg5 = robomath.rotz(math.radians(5))

    # Aplicar rotación acumulativa
    nueva_pose6 = pose_actual6 * rot_5deg6
    nueva_pose5 = pose_actual5 * rot_5deg5

    # Establecer la nueva pose
    frame6.setPose(nueva_pose6)
    frame4.setPose(nueva_pose5)

robot.MoveJ(home_joints)
time.sleep(5.0)

robot.MoveJ(home_joints)
robot.MoveJ(target_poses[0])

RDK.Spray_SetState(SPRAY_ON)

robot.setSpeed(10, 10)
robot.setAcceleration(10)

# Pintado con cambio progresivo de color (10 pasos)
for i, pose in enumerate(target_poses[1:10]):

    actualizar_color(step_index, total_steps)
    robot.MoveJ(pose)
    step_index += 1

# Últimos movimientos

robot.setSpeed(50, 50)
robot.setAcceleration(50)

actualizar_color(step_index, total_steps)
robot.MoveL(target_poses[11])
step_index += 1

# Bucle: 18 pasos de 5 grados
for i in range(18):
    # Obtener la pose actual en cada iteración (actualizada)
    pose_actual6 = frame6.Pose()
    pose_actual5 = frame4.Pose()

    # Crear una rotación de 5 grados en Z
    rot_5deg6 = robomath.rotz(math.radians(5))
    rot_5deg5 = robomath.rotz(math.radians(5))

    # Aplicar rotación acumulativa
    nueva_pose6 = pose_actual6 * rot_5deg6
    nueva_pose5 = pose_actual5 * rot_5deg5

    # Establecer la nueva pose
    frame6.setPose(nueva_pose6)
    frame4.setPose(nueva_pose5)

robot.setSpeed(10, 10)
robot.setAcceleration(10)

for pose in target_poses[12:23]:
    actualizar_color(step_index, total_steps)
    robot.MoveJ(pose)
    step_index += 1

# Bucle: 18 pasos de 5 grados
for i in range(18):
    # Obtener la pose actual en cada iteración (actualizada)
    pose_actual6 = frame6.Pose()
    pose_actual5 = frame4.Pose()

    # Crear una rotación de 5 grados en Z
    rot_5deg6 = robomath.rotz(math.radians(5))
    rot_5deg5 = robomath.rotz(math.radians(5))

    # Aplicar rotación acumulativa
    nueva_pose6 = pose_actual6 * rot_5deg6
    nueva_pose5 = pose_actual5 * rot_5deg5

    # Establecer la nueva pose
    frame6.setPose(nueva_pose6)
    frame4.setPose(nueva_pose5)

for pose in target_poses[23:33]:
    actualizar_color(step_index, total_steps)
    robot.MoveJ(pose)
    step_index += 1

robot.MoveJ(home_joints)

# Bucle: 18 pasos de 5 grados
for i in range(18):
    # Obtener la pose actual en cada iteración (actualizada)
    pose_actual6 = frame6.Pose()
    pose_actual5 = frame4.Pose()

    # Crear una rotación de 5 grados en Z
    rot_5deg6 = robomath.rotz(math.radians(5))
    rot_5deg5 = robomath.rotz(math.radians(5))

    # Aplicar rotación acumulativa
    nueva_pose6 = pose_actual6 * rot_5deg6
    nueva_pose5 = pose_actual5 * rot_5deg5

    # Establecer la nueva pose
    frame6.setPose(nueva_pose6)
    frame4.setPose(nueva_pose5)

for pose in target_poses[33:]:
    actualizar_color(step_index, total_steps)
    robot.MoveJ(pose)
    step_index += 1

robot.MoveJ(home_joints)

# Bucle: 18 pasos de 5 grados
for i in range(18):
    # Obtener la pose actual en cada iteración (actualizada)
    pose_actual6 = frame6.Pose()
    pose_actual5 = frame4.Pose()

    # Crear una rotación de 5 grados en Z
    rot_5deg6 = robomath.rotz(math.radians(5))
    rot_5deg5 = robomath.rotz(math.radians(5))

    # Aplicar rotación acumulativa
    nueva_pose6 = pose_actual6 * rot_5deg6
    nueva_pose5 = pose_actual5 * rot_5deg5

    # Establecer la nueva pose
    frame6.setPose(nueva_pose6)
    frame4.setPose(nueva_pose5)

# Desactivar pintado al finalizar
RDK.Spray_Clear()
RDK.Spray_SetState(SPRAY_OFF)

--- Python program Honda21 ---
from robodk.robolink import *  # API de RoboDK
from robodk.robomath import *  # Funciones matemáticas
import time
import math

# Inicializar conexión con RoboDK
RDK = Robolink()

# Borrar las partículas de pintura previas
RDK.Spray_Clear()

# Comprobar si estamos en modo simulación
if RDK.RunMode() != RUNMODE_SIMULATE:
    raise Exception('El robot no está en modo simulación')

# Obtener el robot
robot = RDK.Item('ABB IRB 580/12S 2', ITEM_TYPE_ROBOT)
if not robot.Valid():
    raise Exception('Robot "ABB IRB 580/12S 2" no encontrado')

# Establecer herramienta activa (TCP2)
tool = RDK.Item('TCP2', ITEM_TYPE_TOOL)
if not tool.Valid():
    raise Exception('Herramienta TCP2 no encontrada')
robot.setTool(tool)

# Obtener el objeto a pintar
obj = RDK.Item('Frame cb 750 1', ITEM_TYPE_OBJECT)
if not obj.Valid():
    raise Exception('Objeto "Frame cb 750 1" no encontrado')

# Obtener el sistema del gancho
frame6 = RDK.Item('Frame H1', ITEM_TYPE_FRAME)
if not frame6.Valid():
    raise Exception('Sistema "Frame H1" no encontrado')

# Obtener el sistema de la honda
frame5 = RDK.Item('Frame 5', ITEM_TYPE_FRAME)
if not frame5.Valid():
    raise Exception('Sistema "Frame 5" no encontrado')

# -------------------------
# MAPEO DE COLORES
# -------------------------
colores_numericos = {
    0: [1.0, 0.0, 0.0],  # rojo
    1: [0.0, 0.0, 0.0],  # negro
    2: [0.0, 1.0, 0.0],  # verde
    3: [0.5, 0.5, 0.5],  # gris
    4: [1.0, 1.0, 1.0],  # blanco
    5: [1.0, 0.5, 0.0]   # naranja
}

# Obtener número desde variable global de RoboDK
valor_color = RDK.getParam('ColorElegido2')
if valor_color is None:
    valor_color = 0  # valor por defecto
valor_color = int(valor_color)

if valor_color not in colores_numericos:
    raise Exception(f'ColorElegido inválido: {valor_color}')
color_final = colores_numericos[valor_color]

# Color neutro inicial
color_inicial = [0.9, 0.9, 0.9]

# Activar pintado automático
options_command = "ELLYPSE PROJECT PARTICLE=SPHERE(4,10,1,1,0.5) STEP=3x3 RAND=2"
close_param = [0, 0, 0, 5, 0, 0, 0, 5, 0, color_final[0], color_final[1], color_final[2], 1]
far_param   = [0, 0, 2000, 500, 0, 2000, 0, 500, 2000, color_final[0], color_final[1], color_final[2], 0.2]
volume = Mat([close_param, far_param]).tr()
RDK.Spray_Add(tool, obj, options_command, volume)
RDK.Spray_SetState(SPRAY_ON)

# Establecer velocidades lentas
robot.setSpeed(50, 50)
robot.setAcceleration(50)

# Lista de nombres de targets
targets = [
    'Pintura21_1',
    'Pintura22_ 1',
    'Pintura22_ 4',
    'Pintura22_ 3',
    'Pintura22_ 2',
    'Pintura22_ 5',
    'Pintura22_ 6',
    'Pintura22_ 7',
    'Pintura22_ 8',
    'Pintura22_ 9',
    'Pintura22_ 10',
    'Pintura22_ 9',
    'Pintura22_ 11',
    'Pintura22_ 9',
    'Pintura21_1',

    'Pintura22_ 12',
    'Pintura22_ 13',
    'Pintura22_ 14',
    'Pintura22_ 15',
    'Pintura22_ 16',
    'Pintura22_ 17',
    'Pintura22_ 18',
    'Pintura22_ 16',
    'Pintura22_ 15',
    'Pintura22_ 14',
    'Pintura22_ 22',
    'Pintura22_ 21',
    'Pintura22_ 23',
    'Pintura22_ 24',
    'Pintura22_ 13',
    'Pintura22_ 19',
    'Pintura22_ 20',
    'Pintura21_1',

    'Pintura22_ 25',
    'Pintura22_ 28',
    'Pintura22_ 27',
    'Pintura22_ 26',
    'Pintura22_ 29',
    'Pintura22_ 30',
    'Pintura22_ 31',
    'Pintura22_ 32',
    'Pintura22_ 33',
    'Pintura22_ 34',
    'Pintura22_ 33',
    'Pintura22_ 35',
    'Pintura22_ 33',
    'Pintura21_1',

    'Pintura22_ 36',
    'Pintura22_ 37',
    'Pintura22_ 38',
    'Pintura22_ 39',
    'Pintura22_ 40',
    'Pintura22_ 41',
    'Pintura22_ 42',
    'Pintura22_ 43',
    'Pintura22_ 44',
    'Pintura22_ 45',
    'Pintura22_ 46',
    'Pintura22_ 47',
    'Pintura22_ 48',
    'Pintura22_ 49',
    'Pintura21_1'


]

# Obtener poses de targets
target_poses = []

# Contar los pasos totales en todas las fases

step_index = 0

# Funcion para actualizar el color de la pieza
def actualizar_color(step_index, total_steps):
    factor = step_index / (total_steps - 1)
    rojo  = color_inicial[0] + (color_final[0] - color_inicial[0]) * factor
    verde = color_inicial[1] + (color_final[1] - color_inicial[1]) * factor
    azul  = color_inicial[2] + (color_final[2] - color_inicial[2]) * factor
    obj.setColor([rojo, verde, azul, 1.0])

for target_name in targets:
    target = RDK.Item(target_name, ITEM_TYPE_TARGET)
    if not target.Valid():
        raise Exception(f'Target no encontrado: {target_name}')
    target_poses.append(target.Pose())

total_steps = len(target_poses)

# Ir a posición de inicio
home_joints = robot.JointsHome()
robot.MoveJ(home_joints)
robot.MoveJ(target_poses[0])

RDK.Spray_SetState(SPRAY_ON)

# Pintado con cambio progresivo de color (10 pasos)
for i, pose in enumerate(target_poses[1:10]):

    actualizar_color(step_index, total_steps)
    robot.MoveL(pose)
    step_index += 1

# Últimos movimientos
robot.setSpeed(50, 50)
robot.setAcceleration(50)
actualizar_color(step_index, total_steps)
robot.MoveL(target_poses[10])
step_index += 1
actualizar_color(step_index, total_steps)
robot.MoveL(target_poses[11])
step_index += 1

robot.setSpeed(10, 10)
robot.setAcceleration(10)
for pose in target_poses[12:15]:
    actualizar_color(step_index, total_steps)
    robot.MoveJ(pose)
    step_index += 1

# Bucle: 18 pasos de 5 grados
for i in range(18):
    # Obtener la pose actual en cada iteración (actualizada)
    pose_actual6 = frame6.Pose()
    pose_actual5 = frame5.Pose()

    # Crear una rotación de 5 grados en Z
    rot_5deg6 = robomath.rotz(math.radians(5))
    rot_5deg5 = robomath.rotz(math.radians(5))

    # Aplicar rotación acumulativa
    nueva_pose6 = pose_actual6 * rot_5deg6
    nueva_pose5 = pose_actual5 * rot_5deg5

    # Establecer la nueva pose
    frame6.setPose(nueva_pose6)
    frame5.setPose(nueva_pose5)

for pose in target_poses[15:29]:
    actualizar_color(step_index, total_steps)
    robot.MoveJ(pose)
    step_index += 1

robot.MoveJ(home_joints)

for pose in target_poses[30:33]:
    actualizar_color(step_index, total_steps)
    robot.MoveJ(pose)
    step_index += 1

# Bucle: 18 pasos de 5 grados
for i in range(18):
    # Obtener la pose actual en cada iteración (actualizada)
    pose_actual6 = frame6.Pose()
    pose_actual5 = frame5.Pose()

    # Crear una rotación de 5 grados en Z
    rot_5deg6 = robomath.rotz(math.radians(5))
    rot_5deg5 = robomath.rotz(math.radians(5))

    # Aplicar rotación acumulativa
    nueva_pose6 = pose_actual6 * rot_5deg6
    nueva_pose5 = pose_actual5 * rot_5deg5

    # Establecer la nueva pose
    frame6.setPose(nueva_pose6)
    frame5.setPose(nueva_pose5)

for pose in target_poses[33:47]:
    actualizar_color(step_index, total_steps)
    robot.MoveJ(pose)
    step_index += 1

# Bucle: 18 pasos de 5 grados
for i in range(18):
    # Obtener la pose actual en cada iteración (actualizada)
    pose_actual6 = frame6.Pose()
    pose_actual5 = frame5.Pose()

    # Crear una rotación de 5 grados en Z
    rot_5deg6 = robomath.rotz(math.radians(5))
    rot_5deg5 = robomath.rotz(math.radians(5))

    # Aplicar rotación acumulativa
    nueva_pose6 = pose_actual6 * rot_5deg6
    nueva_pose5 = pose_actual5 * rot_5deg5

    # Establecer la nueva pose
    frame6.setPose(nueva_pose6)
    frame5.setPose(nueva_pose5)

for pose in target_poses[47:]:
    actualizar_color(step_index, total_steps)
    robot.MoveJ(pose)
    step_index += 1

# Bucle: 18 pasos de 5 grados
for i in range(18):
    # Obtener la pose actual en cada iteración (actualizada)
    pose_actual6 = frame6.Pose()
    pose_actual5 = frame5.Pose()

    # Crear una rotación de 5 grados en Z
    rot_5deg6 = robomath.rotz(math.radians(5))
    rot_5deg5 = robomath.rotz(math.radians(5))

    # Aplicar rotación acumulativa
    nueva_pose6 = pose_actual6 * rot_5deg6
    nueva_pose5 = pose_actual5 * rot_5deg5

    # Establecer la nueva pose
    frame6.setPose(nueva_pose6)
    frame5.setPose(nueva_pose5)

robot.MoveJ(home_joints)
time.sleep(5.0)

robot.MoveJ(home_joints)
robot.MoveJ(target_poses[0])

RDK.Spray_SetState(SPRAY_ON)

# Pintado con cambio progresivo de color (10 pasos)
for i, pose in enumerate(target_poses[1:10]):

    actualizar_color(step_index, total_steps)
    robot.MoveL(pose)
    step_index += 1

# Últimos movimientos
robot.setSpeed(50, 50)
robot.setAcceleration(50)
actualizar_color(step_index, total_steps)
robot.MoveL(target_poses[10])
step_index += 1
actualizar_color(step_index, total_steps)
robot.MoveL(target_poses[11])
step_index += 1

robot.setSpeed(10, 10)
robot.setAcceleration(10)
for pose in target_poses[12:15]:
    actualizar_color(step_index, total_steps)
    robot.MoveJ(pose)
    step_index += 1

# Bucle: 18 pasos de 5 grados
for i in range(18):
    # Obtener la pose actual en cada iteración (actualizada)
    pose_actual6 = frame6.Pose()
    pose_actual5 = frame5.Pose()

    # Crear una rotación de 5 grados en Z
    rot_5deg6 = robomath.rotz(math.radians(5))
    rot_5deg5 = robomath.rotz(math.radians(5))

    # Aplicar rotación acumulativa
    nueva_pose6 = pose_actual6 * rot_5deg6
    nueva_pose5 = pose_actual5 * rot_5deg5

    # Establecer la nueva pose
    frame6.setPose(nueva_pose6)
    frame5.setPose(nueva_pose5)

for pose in target_poses[15:29]:
    actualizar_color(step_index, total_steps)
    robot.MoveJ(pose)
    step_index += 1

robot.MoveJ(home_joints)

for pose in target_poses[30:33]:
    actualizar_color(step_index, total_steps)
    robot.MoveJ(pose)
    step_index += 1

# Bucle: 18 pasos de 5 grados
for i in range(18):
    # Obtener la pose actual en cada iteración (actualizada)
    pose_actual6 = frame6.Pose()
    pose_actual5 = frame5.Pose()

    # Crear una rotación de 5 grados en Z
    rot_5deg6 = robomath.rotz(math.radians(5))
    rot_5deg5 = robomath.rotz(math.radians(5))

    # Aplicar rotación acumulativa
    nueva_pose6 = pose_actual6 * rot_5deg6
    nueva_pose5 = pose_actual5 * rot_5deg5

    # Establecer la nueva pose
    frame6.setPose(nueva_pose6)
    frame5.setPose(nueva_pose5)

for pose in target_poses[33:47]:
    actualizar_color(step_index, total_steps)
    robot.MoveJ(pose)
    step_index += 1

# Bucle: 18 pasos de 5 grados
for i in range(18):
    # Obtener la pose actual en cada iteración (actualizada)
    pose_actual6 = frame6.Pose()
    pose_actual5 = frame5.Pose()

    # Crear una rotación de 5 grados en Z
    rot_5deg6 = robomath.rotz(math.radians(5))
    rot_5deg5 = robomath.rotz(math.radians(5))

    # Aplicar rotación acumulativa
    nueva_pose6 = pose_actual6 * rot_5deg6
    nueva_pose5 = pose_actual5 * rot_5deg5

    # Establecer la nueva pose
    frame6.setPose(nueva_pose6)
    frame5.setPose(nueva_pose5)

for pose in target_poses[47:]:
    actualizar_color(step_index, total_steps)
    robot.MoveJ(pose)
    step_index += 1

# Bucle: 18 pasos de 5 grados
for i in range(18):
    # Obtener la pose actual en cada iteración (actualizada)
    pose_actual6 = frame6.Pose()
    pose_actual5 = frame5.Pose()

    # Crear una rotación de 5 grados en Z
    rot_5deg6 = robomath.rotz(math.radians(5))
    rot_5deg5 = robomath.rotz(math.radians(5))

    # Aplicar rotación acumulativa
    nueva_pose6 = pose_actual6 * rot_5deg6
    nueva_pose5 = pose_actual5 * rot_5deg5

    # Establecer la nueva pose
    frame6.setPose(nueva_pose6)
    frame5.setPose(nueva_pose5)

# Desactivar pintado al finalizar
RDK.Spray_Clear()
RDK.Spray_SetState(SPRAY_OFF)

--- Python program Honda22 ---
from robodk.robolink import *  # API de RoboDK
from robodk.robomath import *  # Funciones matemáticas
import time
import math

# Inicializar conexión con RoboDK
RDK = Robolink()

# Borrar las partículas de pintura previas
RDK.Spray_Clear()

# Comprobar si estamos en modo simulación
if RDK.RunMode() != RUNMODE_SIMULATE:
    raise Exception('El robot no está en modo simulación')

# Obtener el robot
robot = RDK.Item('ABB IRB 580/12S 2', ITEM_TYPE_ROBOT)
if not robot.Valid():
    raise Exception('Robot "ABB IRB 580/12S 2" no encontrado')

# Establecer herramienta activa (TCP2)
tool = RDK.Item('TCP2', ITEM_TYPE_TOOL)
if not tool.Valid():
    raise Exception('Herramienta TCP2 no encontrada')
robot.setTool(tool)

# Obtener el objeto a pintar
obj = RDK.Item('Frame cb 750 2', ITEM_TYPE_OBJECT)
if not obj.Valid():
    raise Exception('Objeto "Frame cb 750 2" no encontrado')

# Obtener el sistema del gancho
frame6 = RDK.Item('Frame H2', ITEM_TYPE_FRAME)
if not frame6.Valid():
    raise Exception('Sistema "Frame H2" no encontrado')

# Obtener el sistema de la honda
frame5 = RDK.Item('Frame 7', ITEM_TYPE_FRAME)
if not frame5.Valid():
    raise Exception('Sistema "Frame 7" no encontrado')

# -------------------------
# MAPEO DE COLORES
# -------------------------
colores_numericos = {
    0: [1.0, 0.0, 0.0],  # rojo
    1: [0.0, 0.0, 0.0],  # negro
    2: [0.0, 1.0, 0.0],  # verde
    3: [0.5, 0.5, 0.5],  # gris
    4: [1.0, 1.0, 1.0],  # blanco
    5: [1.0, 0.5, 0.0]   # naranja
}

# Obtener número desde variable global de RoboDK
valor_color = RDK.getParam('ColorElegido2')
if valor_color is None:
    valor_color = 0  # valor por defecto
valor_color = int(valor_color)

if valor_color not in colores_numericos:
    raise Exception(f'ColorElegido inválido: {valor_color}')
color_final = colores_numericos[valor_color]

# Color neutro inicial
color_inicial = [0.9, 0.9, 0.9]

# Activar pintado automático
options_command = "ELLYPSE PROJECT PARTICLE=SPHERE(4,10,1,1,0.5) STEP=3x3 RAND=2"
close_param = [0, 0, 0, 5, 0, 0, 0, 5, 0, color_final[0], color_final[1], color_final[2], 1]
far_param   = [0, 0, 2000, 500, 0, 2000, 0, 500, 2000, color_final[0], color_final[1], color_final[2], 0.2]
volume = Mat([close_param, far_param]).tr()
RDK.Spray_Add(tool, obj, options_command, volume)
RDK.Spray_SetState(SPRAY_ON)

# Establecer velocidades lentas
robot.setSpeed(50, 50)
robot.setAcceleration(50)

# Lista de nombres de targets
targets = [
    'Pintura21_1',
    'Pintura22_ 1',
    'Pintura22_ 4',
    'Pintura22_ 3',
    'Pintura22_ 2',
    'Pintura22_ 5',
    'Pintura22_ 6',
    'Pintura22_ 7',
    'Pintura22_ 8',
    'Pintura22_ 9',
    'Pintura22_ 10',
    'Pintura22_ 9',
    'Pintura22_ 11',
    'Pintura22_ 9',
    'Pintura21_1',

    'Pintura22_ 12',
    'Pintura22_ 13',
    'Pintura22_ 14',
    'Pintura22_ 15',
    'Pintura22_ 16',
    'Pintura22_ 17',
    'Pintura22_ 18',
    'Pintura22_ 16',
    'Pintura22_ 15',
    'Pintura22_ 14',
    'Pintura22_ 22',
    'Pintura22_ 21',
    'Pintura22_ 23',
    'Pintura22_ 24',
    'Pintura22_ 13',
    'Pintura22_ 19',
    'Pintura22_ 20',
    'Pintura21_1',

    'Pintura22_ 25',
    'Pintura22_ 28',
    'Pintura22_ 27',
    'Pintura22_ 26',
    'Pintura22_ 29',
    'Pintura22_ 30',
    'Pintura22_ 31',
    'Pintura22_ 32',
    'Pintura22_ 33',
    'Pintura22_ 34',
    'Pintura22_ 33',
    'Pintura22_ 35',
    'Pintura22_ 33',
    'Pintura21_1',

    'Pintura22_ 36',
    'Pintura22_ 37',
    'Pintura22_ 38',
    'Pintura22_ 39',
    'Pintura22_ 40',
    'Pintura22_ 41',
    'Pintura22_ 42',
    'Pintura22_ 43',
    'Pintura22_ 44',
    'Pintura22_ 45',
    'Pintura22_ 46',
    'Pintura22_ 47',
    'Pintura22_ 48',
    'Pintura22_ 49',
    'Pintura21_1'


]

# Obtener poses de targets
target_poses = []

# Contar los pasos totales en todas las fases

step_index = 0

